LIN {X 0,Y 520.236,Z 358.517,A -85,B 0,C 180,E1 24281.743,E2 24281.743} C_VEL
LIN {X 0,Y 524.04,Z 361.624,A -85,B 0,C 180,E1 24280.378,E2 24280.378} C_VEL
LIN {X 0,Y 526.654,Z 365.44,A -85,B 0,C 180,E1 24279.437,E2 24279.437} C_VEL
LIN {X 0,Y 529.635,Z 368.07,A -85,B 0,C 180,E1 24278.486,E2 24278.486} C_VEL
LIN {X 0,Y 532.772,Z 372.256,A -85,B 0,C 180,E1 24277.489,E2 24277.489} C_VEL
LIN {X 0,Y 535.113,Z 374.487,A -85,B 0,C 180,E1 24276.809,E2 24276.809} C_VEL
LIN {X 0,Y 538.699,Z 378.866,A -85,B 0,C 180,E1 24275.782,E2 24275.782} C_VEL
LIN {X 0,Y 540.337,Z 380.709,A -85,B 0,C 180,E1 24275.336,E2 24275.336} C_VEL
LIN {X 0,Y 544.251,Z 385.306,A -85,B 0,C 180,E1 24274.305,E2 24274.305} C_VEL
LIN {X 0,Y 549.091,Z 391.188,A -85,B 0,C 180,E1 24273.095,E2 24273.095} C_VEL
LIN {X 0,Y 558.407,Z 402.895,A -85,B 0,C 180,E1 24270.941,E2 24270.941} C_VEL
LIN {X 0,Y 567.449,Z 414.718,A -85,B 0,C 180,E1 24269.034,E2 24269.034} C_VEL
LIN {X 0,Y 578.175,Z 429.194,A -85,B 0,C 180,E1 24266.962,E2 24266.962} C_VEL
LIN {X 0,Y 585.063,Z 439.312,A -85,B 0,C 180,E1 24265.711,E2 24265.711} C_VEL
LIN {X 0,Y 575.969,Z 652.824,A -85,B 0,C 180,E1 24262.521,E2 24262.521} C_VEL
LIN {X 0,Y 569.868,Z 800.136,A -85,B 0,C 180,E1 24260.332,E2 24260.332} C_VEL
LIN {X 0,Y 568.013,Z 824.85,A -85,B 0,C 180,E1 24259.864,E2 24259.864} C_VEL
LIN {X 0,Y 565.088,Z 852.733,A -85,B 0,C 180,E1 24259.144,E2 24259.144} C_VEL
LIN {X 0,Y 562.345,Z 873.984,A -85,B 0,C 180,E1 24258.454,E2 24258.454} C_VEL
LIN {X 0,Y 559.307,Z 894.579,A -85,B 0,C 180,E1 24257.656,E2 24257.656} C_VEL
LIN {X 0,Y 555.969,Z 914.69,A -85,B 0,C 180,E1 24256.747,E2 24256.747} C_VEL
LIN {X 0,Y 551.81,Z 937.435,A -85,B 0,C 180,E1 24255.554,E2 24255.554} C_VEL
LIN {X 0,Y 550.967,Z 941.891,A -85,B 0,C 180,E1 24255.296,E2 24255.296} C_VEL
LIN {X 0,Y 548.862,Z 948.783,A -85,B 0,C 180,E1 24254.955,E2 24254.955} C_VEL
LIN {X 0,Y 540.849,Z 966.119,A -85,B 0,C 180,E1 24254.291,E2 24254.291} C_VEL
LIN {X 0,Y 538.707,Z 972.514,A -85,B 0,C 180,E1 24253.919,E2 24253.919} C_VEL
LIN {X 0,Y 533.191,Z 995.822,A -85,B 0,C 180,E1 24252.097,E2 24252.097} C_VEL
LIN {X 0,Y 528.894,Z 1013.296,A -85,B 0,C 180,E1 24250.536,E2 24250.536} C_VEL
LIN {X 0,Y 524.733,Z 1029.747,A -85,B 0,C 180,E1 24248.891,E2 24248.891} C_VEL
LIN {X 0,Y 520.601,Z 1045.873,A -85,B 0,C 180,E1 24247.089,E2 24247.089} C_VEL
LIN {X 0,Y 515.835,Z 1064.561,A -85,B 0,C 180,E1 24244.741,E2 24244.741} C_VEL
LIN {X 0,Y 511.471,Z 1081.614,A -85,B 0,C 180,E1 24242.254,E2 24242.254} C_VEL
LIN {X 0,Y 508.278,Z 1094.708,A -85,B 0,C 180,E1 24240.107,E2 24240.107} C_VEL
LIN {X 0,Y 505.513,Z 1106.49,A -85,B 0,C 180,E1 24237.954,E2 24237.954} C_VEL
LIN {X 0,Y 502.961,Z 1118.198,A -85,B 0,C 180,E1 24235.555,E2 24235.555} C_VEL
LIN {X 0,Y 500.238,Z 1132.516,A -85,B 0,C 180,E1 24232.195,E2 24232.195} C_VEL
LIN {X 0,Y 498.735,Z 1141.736,A -85,B 0,C 180,E1 24229.682,E2 24229.682} C_VEL
LIN {X 0,Y 497.682,Z 1149.368,A -85,B 0,C 180,E1 24227.298,E2 24227.298} C_VEL
LIN {X 0,Y 496.911,Z 1156.239,A -85,B 0,C 180,E1 24224.806,E2 24224.806} C_VEL
LIN {X 0,Y 496.38,Z 1162.49,A -85,B 0,C 180,E1 24222.092,E2 24222.092} C_VEL
LIN {X 0,Y 496.063,Z 1168.171,A -85,B 0,C 180,E1 24218.928,E2 24218.928} C_VEL
LIN {X 0,Y 495.952,Z 1171.694,A -85,B 0,C 180,E1 24216.134,E2 24216.134} C_VEL
LIN {X 0,Y 495.915,Z 1173.799,A -85,B 0,C 180,E1 24213.578,E2 24213.578} C_VEL
LIN {X 0,Y 495.91,Z 1174.771,A -85,B 0,C 180,E1 24211.155,E2 24211.155} C_VEL
LIN {X 0,Y 495.908,Z 1174.789,A -85,B 0,C 180,E1 24208.845,E2 24208.845} C_VEL
LIN {X 0,Y 495.914,Z 1173.849,A -85,B 0,C 180,E1 24206.417,E2 24206.417} C_VEL
LIN {X 0,Y 495.949,Z 1171.784,A -85,B 0,C 180,E1 24203.866,E2 24203.866} C_VEL
LIN {X 0,Y 496.058,Z 1168.295,A -85,B 0,C 180,E1 24201.072,E2 24201.072} C_VEL
LIN {X 0,Y 496.371,Z 1162.684,A -85,B 0,C 180,E1 24197.908,E2 24197.908} C_VEL
LIN {X 0,Y 496.885,Z 1156.469,A -85,B 0,C 180,E1 24195.194,E2 24195.194} C_VEL
LIN {X 0,Y 497.652,Z 1149.635,A -85,B 0,C 180,E1 24192.701,E2 24192.701} C_VEL
LIN {X 0,Y 498.691,Z 1142.035,A -85,B 0,C 180,E1 24190.316,E2 24190.316} C_VEL
LIN {X 0,Y 500.179,Z 1132.845,A -85,B 0,C 180,E1 24187.802,E2 24187.802} C_VEL
LIN {X 0,Y 502.788,Z 1119.049,A -85,B 0,C 180,E1 24184.538,E2 24184.538} C_VEL
LIN {X 0,Y 505.406,Z 1106.924,A -85,B 0,C 180,E1 24182.04,E2 24182.04} C_VEL
LIN {X 0,Y 508.161,Z 1095.183,A -85,B 0,C 180,E1 24179.885,E2 24179.885} C_VEL
LIN {X 0,Y 511.342,Z 1082.13,A -85,B 0,C 180,E1 24177.737,E2 24177.737} C_VEL
LIN {X 0,Y 515.683,Z 1065.128,A -85,B 0,C 180,E1 24175.247,E2 24175.247} C_VEL
LIN {X 0,Y 520.505,Z 1046.256,A -85,B 0,C 180,E1 24172.865,E2 24172.865} C_VEL
LIN {X 0,Y 524.551,Z 1030.453,A -85,B 0,C 180,E1 24171.093,E2 24171.093} C_VEL
LIN {X 0,Y 528.764,Z 1013.813,A -85,B 0,C 180,E1 24169.422,E2 24169.422} C_VEL
LIN {X 0,Y 533.282,Z 995.499,A -85,B 0,C 180,E1 24167.784,E2 24167.784} C_VEL
LIN {X 0,Y 538.943,Z 971.464,A -85,B 0,C 180,E1 24165.917,E2 24165.917} C_VEL
LIN {X 0,Y 543.469,Z 950.666,A -85,B 0,C 180,E1 24164.528,E2 24164.528} C_VEL
LIN {X 0,Y 547.259,Z 931.938,A -85,B 0,C 180,E1 24163.428,E2 24163.428} C_VEL
LIN {X 0,Y 551.018,Z 911.806,A -85,B 0,C 180,E1 24162.394,E2 24162.394} C_VEL
LIN {X 0,Y 554.725,Z 889.872,A -85,B 0,C 180,E1 24161.426,E2 24161.426} C_VEL
LIN {X 0,Y 558.775,Z 861.74,A -85,B 0,C 180,E1 24160.409,E2 24160.409} C_VEL
LIN {X 0,Y 561.451,Z 839.165,A -85,B 0,C 180,E1 24159.761,E2 24159.761} C_VEL
LIN {X 0,Y 563.504,Z 817.841,A -85,B 0,C 180,E1 24159.27,E2 24159.27} C_VEL
LIN {X 0,Y 565.104,Z 795.465,A -85,B 0,C 180,E1 24158.871,E2 24158.871} C_VEL
LIN {X 0,Y 574.586,Z 574.148,A -85,B 0,C 180,E1 24155.57,E2 24155.57} C_VEL
LIN {X 0,Y 580.415,Z 443.356,A -85,B 0,C 180,E1 24153.594,E2 24153.594} C_VEL
LIN {X 0,Y 568.679,Z 426.867,A -85,B 0,C 180,E1 24151.362,E2 24151.362} C_VEL
LIN {X 0,Y 558.887,Z 413.851,A -85,B 0,C 180,E1 24149.325,E2 24149.325} C_VEL
LIN {X 0,Y 550.085,Z 402.623,A -85,B 0,C 180,E1 24147.321,E2 24147.321} C_VEL
LIN {X 0,Y 545.94,Z 397.535,A -85,B 0,C 180,E1 24146.31,E2 24146.31} C_VEL
LIN {X 0,Y 541.389,Z 391.95,A -85,B 0,C 180,E1 24145.137,E2 24145.137} C_VEL
LIN {X 0,Y 536.861,Z 386.426,A -85,B 0,C 180,E1 24143.897,E2 24143.897} C_VEL
LIN {X 0,Y 533.06,Z 381.8,A -85,B 0,C 180,E1 24142.789,E2 24142.789} C_VEL
LIN {X 0,Y 528.429,Z 376.674,A -85,B 0,C 180,E1 24141.361,E2 24141.361} C_VEL
LIN {X 0,Y 527.196,Z 374.956,A -85,B 0,C 180,E1 24140.948,E2 24140.948} C_VEL
LIN {X 0,Y 523.497,Z 371.232,A -85,B 0,C 180,E1 24139.702,E2 24139.702} C_VEL
LIN {X 0,Y 521.968,Z 368.815,A -85,B 0,C 180,E1 24139.121,E2 24139.121} C_VEL
LIN {X 0,Y 518.399,Z 365.842,A -85,B 0,C 180,E1 24137.801,E2 24137.801} C_VEL
LIN {X 0,Y 516.299,Z 362.399,A -85,B 0,C 180,E1 24136.888,E2 24136.888} C_VEL
LIN {X 0,Y 512.875,Z 359.969,A -85,B 0,C 180,E1 24135.433,E2 24135.433} C_VEL
LIN {X 0,Y 510.92,Z 356.634,A -85,B 0,C 180,E1 24134.42,E2 24134.42} C_VEL
LIN {X 0,Y 510.473,Z 355.792,A -85,B 0,C 180,E1 24134.173,E2 24134.173} C_VEL
LIN {X 0,Y 506.888,Z 353.722,A -85,B 0,C 180,E1 24132.301,E2 24132.301} C_VEL
LIN {X 0,Y 505.032,Z 350.951,A -85,B 0,C 180,E1 24131.072,E2 24131.072} C_VEL
LIN {X 0,Y 504.344,Z 349.04,A -85,B 0,C 180,E1 24130.509,E2 24130.509} C_VEL
LIN {X 0,Y 500.127,Z 346.785,A -85,B 0,C 180,E1 24127.12,E2 24127.12} C_VEL
LIN {X 0,Y 498.094,Z 343.3,A -85,B 0,C 180,E1 24124.144,E2 24124.144} C_VEL
LIN {X 0,Y 497.868,Z 342.14,A -85,B 0,C 180,E1 24123.339,E2 24123.339} C_VEL
LIN {X 0,Y 497.87,Z 342.212,A -85,B 0,C 180,E1 24119.885,E2 24119.885} C_VEL
LIN {X 0,Y 497.933,Z 342.321,A -85,B 0,C 180,E1 24116.777,E2 24116.777} C_VEL
LIN {X 0,Y 498.974,Z 345.261,A -85,B 0,C 180,E1 24114.711,E2 24114.711} C_VEL
LIN {X 0,Y 501.928,Z 348.156,A -85,B 0,C 180,E1 24111.638,E2 24111.638} C_VEL
LIN {X 0,Y 504.476,Z 349.233,A -85,B 0,C 180,E1 24109.811,E2 24109.811} C_VEL
LIN {X 0,Y 505.764,Z 352.251,A -85,B 0,C 180,E1 24108.829,E2 24108.829} C_VEL
LIN {X 0,Y 508.394,Z 354.901,A -85,B 0,C 180,E1 24107.275,E2 24107.275} C_VEL
LIN {X 0,Y 510.655,Z 356.003,A -85,B 0,C 180,E1 24106.15,E2 24106.15} C_VEL
LIN {X 0,Y 512.45,Z 359.379,A -85,B 0,C 180,E1 24105.19,E2 24105.19} C_VEL
LIN {X 0,Y 515.652,Z 362.087,A -85,B 0,C 180,E1 24103.786,E2 24103.786} C_VEL
LIN {X 0,Y 516.704,Z 362.873,A -85,B 0,C 180,E1 24103.357,E2 24103.357} C_VEL
LIN {X 0,Y 519.099,Z 366.62,A -85,B 0,C 180,E1 24102.339,E2 24102.339} C_VEL
LIN {X 0,Y 521.947,Z 369.263,A -85,B 0,C 180,E1 24101.284,E2 24101.284} C_VEL
LIN {X 0,Y 526.752,Z 375.247,A -85,B 0,C 180,E1 24099.586,E2 24099.586} C_VEL
LIN {X 0,Y 531.133,Z 380.666,A -85,B 0,C 180,E1 24098.173,E2 24098.173} C_VEL
LIN {X 0,Y 536.035,Z 386.93,A -85,B 0,C 180,E1 24096.706,E2 24096.706} C_VEL
LIN {X 0,Y 543.551,Z 396.756,A -85,B 0,C 180,E1 24094.649,E2 24094.649} C_VEL
LIN {X 0,Y 552.331,Z 408.685,A -85,B 0,C 180,E1 24092.478,E2 24092.478} C_VEL
LIN {X 0,Y 561.3,Z 421.384,A -85,B 0,C 180,E1 24090.462,E2 24090.462} C_VEL
LIN {X 0,Y 571.815,Z 437.063,A -85,B 0,C 180,E1 24088.3,E2 24088.3} C_VEL
LIN {X 0,Y 580.574,Z 450.913,A -85,B 0,C 180,E1 24086.634,E2 24086.634} C_VEL
LIN {X 0,Y 571.135,Z 666.165,A -85,B 0,C 180,E1 24083.402,E2 24083.402} C_VEL
LIN {X 0,Y 564.461,Z 823.596,A -85,B 0,C 180,E1 24081.051,E2 24081.051} C_VEL
LIN {X 0,Y 562.407,Z 849.401,A -85,B 0,C 180,E1 24080.57,E2 24080.57} C_VEL
LIN {X 0,Y 559.278,Z 877.219,A -85,B 0,C 180,E1 24079.862,E2 24079.862} C_VEL
LIN {X 0,Y 556.351,Z 898.872,A -85,B 0,C 180,E1 24079.166,E2 24079.166} C_VEL
LIN {X 0,Y 553.139,Z 919.668,A -85,B 0,C 180,E1 24078.369,E2 24078.369} C_VEL
LIN {X 0,Y 549.635,Z 940.066,A -85,B 0,C 180,E1 24077.455,E2 24077.455} C_VEL
LIN {X 0,Y 544.928,Z 965.12,A -85,B 0,C 180,E1 24076.145,E2 24076.145} C_VEL
LIN {X 0,Y 539.96,Z 988.657,A -85,B 0,C 180,E1 24074.676,E2 24074.676} C_VEL
LIN {X 0,Y 535.58,Z 1008.335,A -85,B 0,C 180,E1 24073.272,E2 24073.272} C_VEL
LIN {X 0,Y 531.279,Z 1026.905,A -85,B 0,C 180,E1 24071.776,E2 24071.776} C_VEL
LIN {X 0,Y 526.18,Z 1048.396,A -85,B 0,C 180,E1 24069.82,E2 24069.82} C_VEL
LIN {X 0,Y 521.151,Z 1068.846,A -85,B 0,C 180,E1 24067.661,E2 24067.661} C_VEL
LIN {X 0,Y 517.161,Z 1085.154,A -85,B 0,C 180,E1 24065.723,E2 24065.723} C_VEL
LIN {X 0,Y 513.478,Z 1100.386,A -85,B 0,C 180,E1 24063.708,E2 24063.708} C_VEL
LIN {X 0,Y 509.457,Z 1117.58,A -85,B 0,C 180,E1 24061.16,E2 24061.16} C_VEL
LIN {X 0,Y 505.895,Z 1133.58,A -85,B 0,C 180,E1 24058.413,E2 24058.413} C_VEL
LIN {X 0,Y 503.341,Z 1145.834,A -85,B 0,C 180,E1 24056.04,E2 24056.04} C_VEL
LIN {X 0,Y 501.539,Z 1155.249,A -85,B 0,C 180,E1 24053.997,E2 24053.997} C_VEL
LIN {X 0,Y 499.8,Z 1164.972,A -85,B 0,C 180,E1 24051.598,E2 24051.598} C_VEL
LIN {X 0,Y 498.43,Z 1173.911,A -85,B 0,C 180,E1 24049.086,E2 24049.086} C_VEL
LIN {X 0,Y 497.194,Z 1183.627,A -85,B 0,C 180,E1 24045.872,E2 24045.872} C_VEL
LIN {X 0,Y 496.525,Z 1190.553,A -85,B 0,C 180,E1 24043.034,E2 24043.034} C_VEL
LIN {X 0,Y 496.175,Z 1195.689,A -85,B 0,C 180,E1 24040.448,E2 24040.448} C_VEL
LIN {X 0,Y 496.01,Z 1199.512,A -85,B 0,C 180,E1 24037.995,E2 24037.995} C_VEL
LIN {X 0,Y 495.933,Z 1202.422,A -85,B 0,C 180,E1 24035.437,E2 24035.437} C_VEL
LIN {X 0,Y 495.91,Z 1204.435,A -85,B 0,C 180,E1 24032.542,E2 24032.542} C_VEL
LIN {X 0,Y 495.896,Z 1204.894,A -85,B 0,C 180,E1 24029.422,E2 24029.422} C_VEL
LIN {X 0,Y 495.916,Z 1204.094,A -85,B 0,C 180,E1 24026.879,E2 24026.879} C_VEL
LIN {X 0,Y 495.937,Z 1202.193,A -85,B 0,C 180,E1 24024.331,E2 24024.331} C_VEL
LIN {X 0,Y 496.015,Z 1199.351,A -85,B 0,C 180,E1 24021.888,E2 24021.888} C_VEL
LIN {X 0,Y 496.186,Z 1195.48,A -85,B 0,C 180,E1 24019.434,E2 24019.434} C_VEL
LIN {X 0,Y 496.551,Z 1190.298,A -85,B 0,C 180,E1 24016.848,E2 24016.848} C_VEL
LIN {X 0,Y 497.298,Z 1182.679,A -85,B 0,C 180,E1 24013.771,E2 24013.771} C_VEL
LIN {X 0,Y 498.488,Z 1173.505,A -85,B 0,C 180,E1 24010.795,E2 24010.795} C_VEL
LIN {X 0,Y 499.8,Z 1164.976,A -85,B 0,C 180,E1 24008.402,E2 24008.402} C_VEL
LIN {X 0,Y 501.541,Z 1155.256,A -85,B 0,C 180,E1 24006.003,E2 24006.003} C_VEL
LIN {X 0,Y 503.459,Z 1145.256,A -85,B 0,C 180,E1 24003.84,E2 24003.84} C_VEL
LIN {X 0,Y 506.258,Z 1131.902,A -85,B 0,C 180,E1 24001.274,E2 24001.274} C_VEL
LIN {X 0,Y 510.053,Z 1114.954,A -85,B 0,C 180,E1 23998.439,E2 23998.439} C_VEL
LIN {X 0,Y 513.572,Z 1099.989,A -85,B 0,C 180,E1 23996.237,E2 23996.237} C_VEL
LIN {X 0,Y 517.161,Z 1085.156,A -85,B 0,C 180,E1 23994.277,E2 23994.277} C_VEL
LIN {X 0,Y 521.151,Z 1068.847,A -85,B 0,C 180,E1 23992.339,E2 23992.339} C_VEL
LIN {X 0,Y 526.283,Z 1047.928,A -85,B 0,C 180,E1 23990.136,E2 23990.136} C_VEL
LIN {X 0,Y 531.276,Z 1026.894,A -85,B 0,C 180,E1 23988.224,E2 23988.224} C_VEL
LIN {X 0,Y 535.576,Z 1008.328,A -85,B 0,C 180,E1 23986.728,E2 23986.728} C_VEL
LIN {X 0,Y 539.957,Z 988.648,A -85,B 0,C 180,E1 23985.324,E2 23985.324} C_VEL
LIN {X 0,Y 545.113,Z 964.104,A -85,B 0,C 180,E1 23983.8,E2 23983.8} C_VEL
LIN {X 0,Y 549.63,Z 940.037,A -85,B 0,C 180,E1 23982.545,E2 23982.545} C_VEL
LIN {X 0,Y 553.133,Z 919.623,A -85,B 0,C 180,E1 23981.63,E2 23981.63} C_VEL
LIN {X 0,Y 556.346,Z 898.815,A -85,B 0,C 180,E1 23980.833,E2 23980.833} C_VEL
LIN {X 0,Y 559.316,Z 876.821,A -85,B 0,C 180,E1 23980.128,E2 23980.128} C_VEL
LIN {X 0,Y 562.476,Z 848.4,A -85,B 0,C 180,E1 23979.411,E2 23979.411} C_VEL
LIN {X 0,Y 564.452,Z 823.42,A -85,B 0,C 180,E1 23978.948,E2 23978.948} C_VEL
LIN {X 0,Y 572.713,Z 628.453,A -85,B 0,C 180,E1 23976.039,E2 23976.039} C_VEL
LIN {X 0,Y 580.49,Z 450.828,A -85,B 0,C 180,E1 23973.361,E2 23973.361} C_VEL
LIN {X 0,Y 571.078,Z 436.028,A -85,B 0,C 180,E1 23971.568,E2 23971.568} C_VEL
LIN {X 0,Y 560.599,Z 420.343,A -85,B 0,C 180,E1 23969.402,E2 23969.402} C_VEL
LIN {X 0,Y 549.949,Z 405.419,A -85,B 0,C 180,E1 23966.977,E2 23966.977} C_VEL
LIN {X 0,Y 541.131,Z 393.611,A -85,B 0,C 180,E1 23964.741,E2 23964.741} C_VEL
LIN {X 0,Y 534.034,Z 384.385,A -85,B 0,C 180,E1 23962.746,E2 23962.746} C_VEL
LIN {X 0,Y 529.555,Z 378.709,A -85,B 0,C 180,E1 23961.372,E2 23961.372} C_VEL
LIN {X 0,Y 524.876,Z 372.97,A -85,B 0,C 180,E1 23959.822,E2 23959.822} C_VEL
LIN {X 0,Y 521.1,Z 368.313,A -85,B 0,C 180,E1 23958.458,E2 23958.458} C_VEL
LIN {X 0,Y 518.032,Z 365.287,A -85,B 0,C 180,E1 23957.292,E2 23957.292} C_VEL
LIN {X 0,Y 516.304,Z 362.402,A -85,B 0,C 180,E1 23956.54,E2 23956.54} C_VEL
LIN {X 0,Y 512.868,Z 359.866,A -85,B 0,C 180,E1 23955.086,E2 23955.086} C_VEL
LIN {X 0,Y 510.836,Z 356.524,A -85,B 0,C 180,E1 23954.047,E2 23954.047} C_VEL
LIN {X 0,Y 510.437,Z 355.759,A -85,B 0,C 180,E1 23953.827,E2 23953.827} C_VEL
LIN {X 0,Y 507.013,Z 353.838,A -85,B 0,C 180,E1 23952.066,E2 23952.066} C_VEL
LIN {X 0,Y 504.889,Z 350.566,A -85,B 0,C 180,E1 23950.671,E2 23950.671} C_VEL
LIN {X 0,Y 504.421,Z 349.043,A -85,B 0,C 180,E1 23950.277,E2 23950.277} C_VEL
LIN {X 0,Y 500.434,Z 347.063,A -85,B 0,C 180,E1 23947.231,E2 23947.231} C_VEL
LIN {X 0,Y 498.21,Z 343.675,A -85,B 0,C 180,E1 23944.374,E2 23944.374} C_VEL
LIN {X 0,Y 497.91,Z 342.135,A -85,B 0,C 180,E1 23943.569,E2 23943.569} C_VEL
LIN {X 0,Y 497.875,Z 342.216,A -85,B 0,C 180,E1 23940.115,E2 23940.115} C_VEL
LIN {X 0,Y 497.865,Z 342.141,A -85,B 0,C 180,E1 23936.484,E2 23936.484} C_VEL
LIN {X 0,Y 497.918,Z 342.459,A -85,B 0,C 180,E1 23935.797,E2 23935.797} C_VEL
LIN {X 0,Y 499.239,Z 345.748,A -85,B 0,C 180,E1 23933.56,E2 23933.56} C_VEL
LIN {X 0,Y 502.845,Z 348.594,A -85,B 0,C 180,E1 23930.269,E2 23930.269} C_VEL
LIN {X 0,Y 504.501,Z 349.313,A -85,B 0,C 180,E1 23929.147,E2 23929.147} C_VEL
LIN {X 0,Y 505.68,Z 352.253,A -85,B 0,C 180,E1 23928.249,E2 23928.249} C_VEL
LIN {X 0,Y 508.557,Z 354.98,A -85,B 0,C 180,E1 23926.585,E2 23926.585} C_VEL
LIN {X 0,Y 510.678,Z 356.028,A -85,B 0,C 180,E1 23925.544,E2 23925.544} C_VEL
LIN {X 0,Y 512.428,Z 359.427,A -85,B 0,C 180,E1 23924.611,E2 23924.611} C_VEL
LIN {X 0,Y 515.393,Z 361.958,A -85,B 0,C 180,E1 23923.314,E2 23923.314} C_VEL
LIN {X 0,Y 516.584,Z 362.81,A -85,B 0,C 180,E1 23922.832,E2 23922.832} C_VEL
LIN {X 0,Y 518.994,Z 366.518,A -85,B 0,C 180,E1 23921.814,E2 23921.814} C_VEL
LIN {X 0,Y 522.327,Z 369.303,A -85,B 0,C 180,E1 23920.602,E2 23920.602} C_VEL
LIN {X 0,Y 525.385,Z 373.462,A -85,B 0,C 180,E1 23919.501,E2 23919.501} C_VEL
LIN {X 0,Y 527.855,Z 375.748,A -85,B 0,C 180,E1 23918.702,E2 23918.702} C_VEL
LIN {X 0,Y 531.312,Z 380.127,A -85,B 0,C 180,E1 23917.599,E2 23917.599} C_VEL
LIN {X 0,Y 533.271,Z 382.147,A -85,B 0,C 180,E1 23917.018,E2 23917.018} C_VEL
LIN {X 0,Y 537.21,Z 386.738,A -85,B 0,C 180,E1 23915.886,E2 23915.886} C_VEL
LIN {X 0,Y 542.151,Z 392.676,A -85,B 0,C 180,E1 23914.55,E2 23914.55} C_VEL
LIN {X 0,Y 546.944,Z 398.552,A -85,B 0,C 180,E1 23913.333,E2 23913.333} C_VEL
LIN {X 0,Y 556.267,Z 410.523,A -85,B 0,C 180,E1 23911.143,E2 23911.143} C_VEL
LIN {X 0,Y 564.469,Z 421.296,A -85,B 0,C 180,E1 23909.384,E2 23909.384} C_VEL
LIN {X 0,Y 575.542,Z 436.424,A -85,B 0,C 180,E1 23907.207,E2 23907.207} C_VEL
LIN {X 0,Y 580.401,Z 443.667,A -85,B 0,C 180,E1 23906.303,E2 23906.303} C_VEL
LIN {X 0,Y 570.968,Z 656.962,A -85,B 0,C 180,E1 23903.101,E2 23903.101} C_VEL
LIN {X 0,Y 564.79,Z 800.458,A -85,B 0,C 180,E1 23900.956,E2 23900.956} C_VEL
LIN {X 0,Y 562.856,Z 825.404,A -85,B 0,C 180,E1 23900.482,E2 23900.482} C_VEL
LIN {X 0,Y 559.848,Z 853.118,A -85,B 0,C 180,E1 23899.763,E2 23899.763} C_VEL
LIN {X 0,Y 556.979,Z 874.623,A -85,B 0,C 180,E1 23899.061,E2 23899.061} C_VEL
LIN {X 0,Y 553.916,Z 894.727,A -85,B 0,C 180,E1 23898.279,E2 23898.279} C_VEL
LIN {X 0,Y 550.349,Z 915.483,A -85,B 0,C 180,E1 23897.337,E2 23897.337} C_VEL
LIN {X 0,Y 545.768,Z 939.703,A -85,B 0,C 180,E1 23896.053,E2 23896.053} C_VEL
LIN {X 0,Y 540.731,Z 963.237,A -85,B 0,C 180,E1 23894.566,E2 23894.566} C_VEL
LIN {X 0,Y 538.707,Z 972.514,A -85,B 0,C 180,E1 23893.919,E2 23893.919} C_VEL
LIN {X 0,Y 536.517,Z 978.993,A -85,B 0,C 180,E1 23893.526,E2 23893.526} C_VEL
LIN {X 0,Y 528.001,Z 995.476,A -85,B 0,C 180,E1 23892.675,E2 23892.675} C_VEL
LIN {X 0,Y 525.705,Z 1001.573,A -85,B 0,C 180,E1 23892.226,E2 23892.226} C_VEL
LIN {X 0,Y 520.245,Z 1022.906,A -85,B 0,C 180,E1 23890.222,E2 23890.222} C_VEL
LIN {X 0,Y 515.074,Z 1042.157,A -85,B 0,C 180,E1 23888.119,E2 23888.119} C_VEL
LIN {X 0,Y 510.918,Z 1057.554,A -85,B 0,C 180,E1 23886.228,E2 23886.228} C_VEL
LIN {X 0,Y 507.147,Z 1071.643,A -85,B 0,C 180,E1 23884.299,E2 23884.299} C_VEL
LIN {X 0,Y 503.464,Z 1085.677,A -85,B 0,C 180,E1 23882.157,E2 23882.157} C_VEL
LIN {X 0,Y 499.39,Z 1101.788,A -85,B 0,C 180,E1 23879.375,E2 23879.375} C_VEL
LIN {X 0,Y 496.221,Z 1115.105,A -85,B 0,C 180,E1 23876.701,E2 23876.701} C_VEL
LIN {X 0,Y 493.89,Z 1125.827,A -85,B 0,C 180,E1 23874.265,E2 23874.265} C_VEL
LIN {X 0,Y 492.03,Z 1135.294,A -85,B 0,C 180,E1 23871.831,E2 23871.831} C_VEL
LIN {X 0,Y 490.343,Z 1145.785,A -85,B 0,C 180,E1 23868.795,E2 23868.795} C_VEL
LIN {X 0,Y 489.167,Z 1154.722,A -85,B 0,C 180,E1 23865.653,E2 23865.653} C_VEL
LIN {X 0,Y 488.537,Z 1160.963,A -85,B 0,C 180,E1 23863.01,E2 23863.01} C_VEL
LIN {X 0,Y 488.194,Z 1165.812,A -85,B 0,C 180,E1 23860.502,E2 23860.502} C_VEL
LIN {X 0,Y 488.016,Z 1169.607,A -85,B 0,C 180,E1 23858.008,E2 23858.008} C_VEL
LIN {X 0,Y 487.932,Z 1172.488,A -85,B 0,C 180,E1 23855.409,E2 23855.409} C_VEL
LIN {X 0,Y 487.908,Z 1174.529,A -85,B 0,C 180,E1 23852.349,E2 23852.349} C_VEL
LIN {X 0,Y 487.898,Z 1174.88,A -85,B 0,C 180,E1 23849.295,E2 23849.295} C_VEL
LIN {X 0,Y 487.912,Z 1174.05,A -85,B 0,C 180,E1 23846.711,E2 23846.711} C_VEL
LIN {X 0,Y 487.939,Z 1172.235,A -85,B 0,C 180,E1 23844.237,E2 23844.237} C_VEL
LIN {X 0,Y 488.027,Z 1169.374,A -85,B 0,C 180,E1 23841.728,E2 23841.728} C_VEL
LIN {X 0,Y 488.205,Z 1165.555,A -85,B 0,C 180,E1 23839.259,E2 23839.259} C_VEL
LIN {X 0,Y 488.598,Z 1160.39,A -85,B 0,C 180,E1 23836.63,E2 23836.63} C_VEL
LIN {X 0,Y 489.392,Z 1152.808,A -85,B 0,C 180,E1 23833.502,E2 23833.502} C_VEL
LIN {X 0,Y 490.647,Z 1143.652,A -85,B 0,C 180,E1 23830.476,E2 23830.476} C_VEL
LIN {X 0,Y 492.222,Z 1134.266,A -85,B 0,C 180,E1 23827.801,E2 23827.801} C_VEL
LIN {X 0,Y 494.233,Z 1124.162,A -85,B 0,C 180,E1 23825.243,E2 23825.243} C_VEL
LIN {X 0,Y 497.333,Z 1110.308,A -85,B 0,C 180,E1 23822.198,E2 23822.198} C_VEL
LIN {X 0,Y 500.633,Z 1096.75,A -85,B 0,C 180,E1 23819.634,E2 23819.634} C_VEL
LIN {X 0,Y 503.904,Z 1083.914,A -85,B 0,C 180,E1 23817.471,E2 23817.471} C_VEL
LIN {X 0,Y 507.473,Z 1070.386,A -85,B 0,C 180,E1 23815.428,E2 23815.428} C_VEL
LIN {X 0,Y 512.006,Z 1053.586,A -85,B 0,C 180,E1 23813.165,E2 23813.165} C_VEL
LIN {X 0,Y 517.43,Z 1033.343,A -85,B 0,C 180,E1 23810.796,E2 23810.796} C_VEL
LIN {X 0,Y 521.878,Z 1016.482,A -85,B 0,C 180,E1 23809.063,E2 23809.063} C_VEL
LIN {X 0,Y 526.393,Z 998.904,A -85,B 0,C 180,E1 23807.452,E2 23807.452} C_VEL
LIN {X 0,Y 531.06,Z 980.034,A -85,B 0,C 180,E1 23805.919,E2 23805.919} C_VEL
LIN {X 0,Y 536.817,Z 955.391,A -85,B 0,C 180,E1 23804.186,E2 23804.186} C_VEL
LIN {X 0,Y 541.294,Z 934.192,A -85,B 0,C 180,E1 23802.912,E2 23802.912} C_VEL
LIN {X 0,Y 545.165,Z 914.308,A -85,B 0,C 180,E1 23801.874,E2 23801.874} C_VEL
LIN {X 0,Y 548.546,Z 895.233,A -85,B 0,C 180,E1 23801.009,E2 23801.009} C_VEL
LIN {X 0,Y 551.825,Z 874.442,A -85,B 0,C 180,E1 23800.199,E2 23800.199} C_VEL
LIN {X 0,Y 555.076,Z 850.656,A -85,B 0,C 180,E1 23799.429,E2 23799.429} C_VEL
LIN {X 0,Y 558.081,Z 822.454,A -85,B 0,C 180,E1 23798.723,E2 23798.723} C_VEL
LIN {X 0,Y 559.878,Z 799.571,A -85,B 0,C 180,E1 23798.296,E2 23798.296} C_VEL
LIN {X 0,Y 569.203,Z 591.089,A -85,B 0,C 180,E1 23795.167,E2 23795.167} C_VEL
LIN {X 0,Y 575.765,Z 447.836,A -85,B 0,C 180,E1 23792.986,E2 23792.986} C_VEL
LIN {X 0,Y 565.116,Z 432.652,A -85,B 0,C 180,E1 23790.901,E2 23790.901} C_VEL
LIN {X 0,Y 555.679,Z 420.101,A -85,B 0,C 180,E1 23788.891,E2 23788.891} C_VEL
LIN {X 0,Y 547.618,Z 409.649,A -85,B 0,C 180,E1 23787.013,E2 23787.013} C_VEL
LIN {X 0,Y 543.33,Z 404.368,A -85,B 0,C 180,E1 23785.947,E2 23785.947} C_VEL
LIN {X 0,Y 539.124,Z 399.122,A -85,B 0,C 180,E1 23784.84,E2 23784.84} C_VEL
LIN {X 0,Y 534.653,Z 393.631,A -85,B 0,C 180,E1 23783.592,E2 23783.592} C_VEL
LIN {X 0,Y 530.064,Z 388.145,A -85,B 0,C 180,E1 23782.223,E2 23782.223} C_VEL
LIN {X 0,Y 526.282,Z 383.698,A -85,B 0,C 180,E1 23781.015,E2 23781.015} C_VEL
LIN {X 0,Y 525.123,Z 382.294,A -85,B 0,C 180,E1 23780.626,E2 23780.626} C_VEL
LIN {X 0,Y 521.441,Z 378.283,A -85,B 0,C 180,E1 23779.345,E2 23779.345} C_VEL
LIN {X 0,Y 520.128,Z 376.353,A -85,B 0,C 180,E1 23778.842,E2 23778.842} C_VEL
LIN {X 0,Y 516.637,Z 373.217,A -85,B 0,C 180,E1 23777.515,E2 23777.515} C_VEL
LIN {X 0,Y 514.815,Z 370.16,A -85,B 0,C 180,E1 23776.705,E2 23776.705} C_VEL
LIN {X 0,Y 511.442,Z 367.658,A -85,B 0,C 180,E1 23775.245,E2 23775.245} C_VEL
LIN {X 0,Y 509.313,Z 364.016,A -85,B 0,C 180,E1 23774.119,E2 23774.119} C_VEL
LIN {X 0,Y 508.386,Z 363.363,A -85,B 0,C 180,E1 23773.652,E2 23773.652} C_VEL
LIN {X 0,Y 504.835,Z 360.625,A -85,B 0,C 180,E1 23771.655,E2 23771.655} C_VEL
LIN {X 0,Y 503.288,Z 357.422,A -85,B 0,C 180,E1 23770.503,E2 23770.503} C_VEL
LIN {X 0,Y 502.87,Z 356.873,A -85,B 0,C 180,E1 23770.193,E2 23770.193} C_VEL
LIN {X 0,Y 498.944,Z 354.543,A -85,B 0,C 180,E1 23766.906,E2 23766.906} C_VEL
LIN {X 0,Y 497.062,Z 351.182,A -85,B 0,C 180,E1 23764.037,E2 23764.037} C_VEL
LIN {X 0,Y 496.78,Z 350.063,A -85,B 0,C 180,E1 23763.231,E2 23763.231} C_VEL
LIN {X 0,Y 496.906,Z 350.216,A -85,B 0,C 180,E1 23756.886,E2 23756.886} C_VEL
LIN {X 0,Y 497.916,Z 353.139,A -85,B 0,C 180,E1 23754.815,E2 23754.815} C_VEL
LIN {X 0,Y 500.822,Z 356.043,A -85,B 0,C 180,E1 23751.735,E2 23751.735} C_VEL
LIN {X 0,Y 503.202,Z 357.18,A -85,B 0,C 180,E1 23749.987,E2 23749.987} C_VEL
LIN {X 0,Y 504.78,Z 360.426,A -85,B 0,C 180,E1 23748.806,E2 23748.806} C_VEL
LIN {X 0,Y 507.437,Z 362.898,A -85,B 0,C 180,E1 23747.25,E2 23747.25} C_VEL
LIN {X 0,Y 509.233,Z 363.883,A -85,B 0,C 180,E1 23746.343,E2 23746.343} C_VEL
LIN {X 0,Y 511.359,Z 367.473,A -85,B 0,C 180,E1 23745.216,E2 23745.216} C_VEL
LIN {X 0,Y 515.143,Z 370.63,A -85,B 0,C 180,E1 23743.567,E2 23743.567} C_VEL
LIN {X 0,Y 517.859,Z 374.597,A -85,B 0,C 180,E1 23742.412,E2 23742.412} C_VEL
LIN {X 0,Y 520.261,Z 376.826,A -85,B 0,C 180,E1 23741.511,E2 23741.511} C_VEL
LIN {X 0,Y 525.003,Z 382.828,A -85,B 0,C 180,E1 23739.806,E2 23739.806} C_VEL
LIN {X 0,Y 529.251,Z 388.167,A -85,B 0,C 180,E1 23738.412,E2 23738.412} C_VEL
LIN {X 0,Y 534.011,Z 394.317,A -85,B 0,C 180,E1 23736.962,E2 23736.962} C_VEL
LIN {X 0,Y 541.346,Z 404.043,A -85,B 0,C 180,E1 23734.919,E2 23734.919} C_VEL
LIN {X 0,Y 550.432,Z 416.532,A -85,B 0,C 180,E1 23732.639,E2 23732.639} C_VEL
LIN {X 0,Y 559.972,Z 430.331,A -85,B 0,C 180,E1 23730.473,E2 23730.473} C_VEL
LIN {X 0,Y 570.34,Z 446.124,A -85,B 0,C 180,E1 23728.327,E2 23728.327} C_VEL
LIN {X 0,Y 575.955,Z 455.358,A -85,B 0,C 180,E1 23727.232,E2 23727.232} C_VEL
LIN {X 0,Y 566.218,Z 669.367,A -85,B 0,C 180,E1 23724.004,E2 23724.004} C_VEL
LIN {X 0,Y 559.434,Z 823.349,A -85,B 0,C 180,E1 23721.692,E2 23721.692} C_VEL
LIN {X 0,Y 557.308,Z 849.313,A -85,B 0,C 180,E1 23721.207,E2 23721.207} C_VEL
LIN {X 0,Y 554.093,Z 876.962,A -85,B 0,C 180,E1 23720.502,E2 23720.502} C_VEL
LIN {X 0,Y 551.068,Z 898.613,A -85,B 0,C 180,E1 23719.806,E2 23719.806} C_VEL
LIN {X 0,Y 547.746,Z 919.406,A -85,B 0,C 180,E1 23719.008,E2 23719.008} C_VEL
LIN {X 0,Y 544.122,Z 939.802,A -85,B 0,C 180,E1 23718.091,E2 23718.091} C_VEL
LIN {X 0,Y 539.247,Z 964.854,A -85,B 0,C 180,E1 23716.776,E2 23716.776} C_VEL
LIN {X 0,Y 534.018,Z 988.721,A -85,B 0,C 180,E1 23715.279,E2 23715.279} C_VEL
LIN {X 0,Y 529.488,Z 1008.324,A -85,B 0,C 180,E1 23713.87,E2 23713.87} C_VEL
LIN {X 0,Y 524.993,Z 1026.966,A -85,B 0,C 180,E1 23712.355,E2 23712.355} C_VEL
LIN {X 0,Y 519.61,Z 1048.704,A -85,B 0,C 180,E1 23710.356,E2 23710.356} C_VEL
LIN {X 0,Y 514.366,Z 1069.042,A -85,B 0,C 180,E1 23708.181,E2 23708.181} C_VEL
LIN {X 0,Y 510.251,Z 1085.136,A -85,B 0,C 180,E1 23706.245,E2 23706.245} C_VEL
LIN {X 0,Y 506.456,Z 1100.108,A -85,B 0,C 180,E1 23704.239,E2 23704.239} C_VEL
LIN {X 0,Y 502.318,Z 1117.027,A -85,B 0,C 180,E1 23701.701,E2 23701.701} C_VEL
LIN {X 0,Y 498.513,Z 1133.144,A -85,B 0,C 180,E1 23698.906,E2 23698.906} C_VEL
LIN {X 0,Y 495.795,Z 1145.558,A -85,B 0,C 180,E1 23696.467,E2 23696.467} C_VEL
LIN {X 0,Y 493.69,Z 1156.076,A -85,B 0,C 180,E1 23694.149,E2 23694.149} C_VEL
LIN {X 0,Y 491.913,Z 1165.888,A -85,B 0,C 180,E1 23691.711,E2 23691.711} C_VEL
LIN {X 0,Y 490.276,Z 1176.321,A -85,B 0,C 180,E1 23688.674,E2 23688.674} C_VEL
LIN {X 0,Y 489.153,Z 1184.836,A -85,B 0,C 180,E1 23685.653,E2 23685.653} C_VEL
LIN {X 0,Y 488.553,Z 1190.804,A -85,B 0,C 180,E1 23683.13,E2 23683.13} C_VEL
LIN {X 0,Y 488.196,Z 1195.684,A -85,B 0,C 180,E1 23680.622,E2 23680.622} C_VEL
LIN {X 0,Y 488.017,Z 1199.509,A -85,B 0,C 180,E1 23678.127,E2 23678.127} C_VEL
LIN {X 0,Y 487.937,Z 1202.305,A -85,B 0,C 180,E1 23675.645,E2 23675.645} C_VEL
LIN {X 0,Y 487.914,Z 1204.228,A -85,B 0,C 180,E1 23672.937,E2 23672.937} C_VEL
LIN {X 0,Y 487.9,Z 1204.961,A -85,B 0,C 180,E1 23669.765,E2 23669.765} C_VEL
LIN {X 0,Y 487.916,Z 1204.091,A -85,B 0,C 180,E1 23666.828,E2 23666.828} C_VEL
LIN {X 0,Y 487.939,Z 1202.19,A -85,B 0,C 180,E1 23664.237,E2 23664.237} C_VEL
LIN {X 0,Y 488.022,Z 1199.318,A -85,B 0,C 180,E1 23661.732,E2 23661.732} C_VEL
LIN {X 0,Y 488.206,Z 1195.477,A -85,B 0,C 180,E1 23659.259,E2 23659.259} C_VEL
LIN {X 0,Y 488.605,Z 1190.295,A -85,B 0,C 180,E1 23656.63,E2 23656.63} C_VEL
LIN {X 0,Y 489.406,Z 1182.678,A -85,B 0,C 180,E1 23653.502,E2 23653.502} C_VEL
LIN {X 0,Y 490.674,Z 1173.504,A -85,B 0,C 180,E1 23650.477,E2 23650.477} C_VEL
LIN {X 0,Y 492.077,Z 1164.966,A -85,B 0,C 180,E1 23648.045,E2 23648.045} C_VEL
LIN {X 0,Y 493.889,Z 1155.031,A -85,B 0,C 180,E1 23645.607,E2 23645.607} C_VEL
LIN {X 0,Y 496.185,Z 1143.81,A -85,B 0,C 180,E1 23643.168,E2 23643.168} C_VEL
LIN {X 0,Y 499.588,Z 1128.516,A -85,B 0,C 180,E1 23640.242,E2 23640.242} C_VEL
LIN {X 0,Y 503.247,Z 1113.109,A -85,B 0,C 180,E1 23637.693,E2 23637.693} C_VEL
LIN {X 0,Y 506.807,Z 1098.658,A -85,B 0,C 180,E1 23635.557,E2 23635.557} C_VEL
LIN {X 0,Y 510.791,Z 1082.998,A -85,B 0,C 180,E1 23633.482,E2 23633.482} C_VEL
LIN {X 0,Y 516.011,Z 1062.79,A -85,B 0,C 180,E1 23631.112,E2 23631.112} C_VEL
LIN {X 0,Y 520.963,Z 1043.19,A -85,B 0,C 180,E1 23629.121,E2 23629.121} C_VEL
LIN {X 0,Y 525.407,Z 1025.267,A -85,B 0,C 180,E1 23627.502,E2 23627.502} C_VEL
LIN {X 0,Y 529.846,Z 1006.816,A -85,B 0,C 180,E1 23626.017,E2 23626.017} C_VEL
LIN {X 0,Y 534.804,Z 985.357,A -85,B 0,C 180,E1 23624.495,E2 23624.495} C_VEL
LIN {X 0,Y 540.241,Z 959.776,A -85,B 0,C 180,E1 23622.948,E2 23622.948} C_VEL
LIN {X 0,Y 544.326,Z 938.622,A -85,B 0,C 180,E1 23621.854,E2 23621.854} C_VEL
LIN {X 0,Y 547.957,Z 918.056,A -85,B 0,C 180,E1 23620.938,E2 23620.938} C_VEL
LIN {X 0,Y 551.286,Z 897.053,A -85,B 0,C 180,E1 23620.141,E2 23620.141} C_VEL
LIN {X 0,Y 554.958,Z 870.498,A -85,B 0,C 180,E1 23619.312,E2 23619.312} C_VEL
LIN {X 0,Y 557.735,Z 844.278,A -85,B 0,C 180,E1 23618.694,E2 23618.694} C_VEL
LIN {X 0,Y 559.513,Z 821.634,A -85,B 0,C 180,E1 23618.282,E2 23618.282} C_VEL
LIN {X 0,Y 568.788,Z 610.555,A -85,B 0,C 180,E1 23615.116,E2 23615.116} C_VEL
LIN {X 0,Y 575.874,Z 454.996,A -85,B 0,C 180,E1 23612.757,E2 23612.757} C_VEL
LIN {X 0,Y 564.913,Z 437.802,A -85,B 0,C 180,E1 23610.589,E2 23610.589} C_VEL
LIN {X 0,Y 556.614,Z 425.504,A -85,B 0,C 180,E1 23608.808,E2 23608.808} C_VEL
LIN {X 0,Y 547.474,Z 412.435,A -85,B 0,C 180,E1 23606.669,E2 23606.669} C_VEL
LIN {X 0,Y 538.68,Z 400.519,A -85,B 0,C 180,E1 23604.394,E2 23604.394} C_VEL
LIN {X 0,Y 532.034,Z 391.747,A -85,B 0,C 180,E1 23602.486,E2 23602.486} C_VEL
LIN {X 0,Y 527.45,Z 385.914,A -85,B 0,C 180,E1 23601.053,E2 23601.053} C_VEL
LIN {X 0,Y 523.001,Z 380.344,A -85,B 0,C 180,E1 23599.547,E2 23599.547} C_VEL
LIN {X 0,Y 519.417,Z 375.916,A -85,B 0,C 180,E1 23598.229,E2 23598.229} C_VEL
LIN {X 0,Y 516.271,Z 372.648,A -85,B 0,C 180,E1 23597.005,E2 23597.005} C_VEL
LIN {X 0,Y 514.816,Z 370.159,A -85,B 0,C 180,E1 23596.357,E2 23596.357} C_VEL
LIN {X 0,Y 511.316,Z 367.421,A -85,B 0,C 180,E1 23594.843,E2 23594.843} C_VEL
LIN {X 0,Y 509.223,Z 363.899,A -85,B 0,C 180,E1 23593.744,E2 23593.744} C_VEL
LIN {X 0,Y 505.208,Z 361.026,A -85,B 0,C 180,E1 23591.589,E2 23591.589} C_VEL
LIN {X 0,Y 503.303,Z 357.543,A -85,B 0,C 180,E1 23590.242,E2 23590.242} C_VEL
LIN {X 0,Y 502.936,Z 356.865,A -85,B 0,C 180,E1 23589.96,E2 23589.96} C_VEL
LIN {X 0,Y 499.003,Z 354.649,A -85,B 0,C 180,E1 23586.79,E2 23586.79} C_VEL
LIN {X 0,Y 496.962,Z 350.768,A -85,B 0,C 180,E1 23583.807,E2 23583.807} C_VEL
LIN {X 0,Y 496.783,Z 350.052,A -85,B 0,C 180,E1 23583.346,E2 23583.346} C_VEL
LIN {X 0,Y 496.819,Z 350.079,A -85,B 0,C 180,E1 23576.076,E2 23576.076} C_VEL
LIN {X 0,Y 498.17,Z 353.626,A -85,B 0,C 180,E1 23573.662,E2 23573.662} C_VEL
LIN {X 0,Y 501.726,Z 356.486,A -85,B 0,C 180,E1 23570.363,E2 23570.363} C_VEL
LIN {X 0,Y 503.188,Z 357.178,A -85,B 0,C 180,E1 23569.35,E2 23569.35} C_VEL
LIN {X 0,Y 504.611,Z 360.322,A -85,B 0,C 180,E1 23568.281,E2 23568.281} C_VEL
LIN {X 0,Y 508.034,Z 363.206,A -85,B 0,C 180,E1 23566.339,E2 23566.339} C_VEL
LIN {X 0,Y 509.251,Z 363.934,A -85,B 0,C 180,E1 23565.735,E2 23565.735} C_VEL
LIN {X 0,Y 511.336,Z 367.543,A -85,B 0,C 180,E1 23564.635,E2 23564.635} C_VEL
LIN {X 0,Y 515.022,Z 370.571,A -85,B 0,C 180,E1 23563.04,E2 23563.04} C_VEL
LIN {X 0,Y 517.62,Z 374.352,A -85,B 0,C 180,E1 23561.938,E2 23561.938} C_VEL
LIN {X 0,Y 520.693,Z 377.065,A -85,B 0,C 180,E1 23560.801,E2 23560.801} C_VEL
LIN {X 0,Y 523.964,Z 381.309,A -85,B 0,C 180,E1 23559.618,E2 23559.618} C_VEL
LIN {X 0,Y 526.087,Z 383.392,A -85,B 0,C 180,E1 23558.919,E2 23558.919} C_VEL
LIN {X 0,Y 529.856,Z 387.981,A -85,B 0,C 180,E1 23557.709,E2 23557.709} C_VEL
LIN {X 0,Y 531.533,Z 389.92,A -85,B 0,C 180,E1 23557.2,E2 23557.2} C_VEL
LIN {X 0,Y 536.399,Z 395.783,A -85,B 0,C 180,E1 23555.789,E2 23555.789} C_VEL
LIN {X 0,Y 541.248,Z 401.786,A -85,B 0,C 180,E1 23554.475,E2 23554.475} C_VEL
LIN {X 0,Y 546.539,Z 408.356,A -85,B 0,C 180,E1 23553.135,E2 23553.135} C_VEL
LIN {X 0,Y 553.314,Z 416.958,A -85,B 0,C 180,E1 23551.535,E2 23551.535} C_VEL
LIN {X 0,Y 562.606,Z 429.371,A -85,B 0,C 180,E1 23549.509,E2 23549.509} C_VEL
LIN {X 0,Y 573.617,Z 444.659,A -85,B 0,C 180,E1 23547.321,E2 23547.321} C_VEL
LIN {X 0,Y 575.795,Z 448.147,A -85,B 0,C 180,E1 23546.902,E2 23546.902} C_VEL
LIN {X 0,Y 566.004,Z 661.624,A -85,B 0,C 180,E1 23543.683,E2 23543.683} C_VEL
LIN {X 0,Y 559.781,Z 800.774,A -85,B 0,C 180,E1 23541.592,E2 23541.592} C_VEL
LIN {X 0,Y 557.769,Z 825.938,A -85,B 0,C 180,E1 23541.112,E2 23541.112} C_VEL
LIN {X 0,Y 554.675,Z 853.503,A -85,B 0,C 180,E1 23540.393,E2 23540.393} C_VEL
LIN {X 0,Y 551.68,Z 875.247,A -85,B 0,C 180,E1 23539.681,E2 23539.681} C_VEL
LIN {X 0,Y 548.57,Z 895.002,A -85,B 0,C 180,E1 23538.909,E2 23538.909} C_VEL
LIN {X 0,Y 544.98,Z 915.222,A -85,B 0,C 180,E1 23537.991,E2 23537.991} C_VEL
LIN {X 0,Y 540.527,Z 937.986,A -85,B 0,C 180,E1 23536.787,E2 23536.787} C_VEL
LIN {X 0,Y 535,Z 963.2,A -85,B 0,C 180,E1 23535.203,E2 23535.203} C_VEL
LIN {X 0,Y 530.368,Z 982.768,A -85,B 0,C 180,E1 23533.778,E2 23533.778} C_VEL
LIN {X 0,Y 525.92,Z 1000.719,A -85,B 0,C 180,E1 23532.3,E2 23532.3} C_VEL
LIN {X 0,Y 525.705,Z 1001.573,A -85,B 0,C 180,E1 23532.226,E2 23532.226} C_VEL
LIN {X 0,Y 523.433,Z 1007.72,A -85,B 0,C 180,E1 23531.764,E2 23531.764} C_VEL
LIN {X 0,Y 514.264,Z 1024.108,A -85,B 0,C 180,E1 23530.662,E2 23530.662} C_VEL
LIN {X 0,Y 512.332,Z 1028.898,A -85,B 0,C 180,E1 23530.207,E2 23530.207} C_VEL
LIN {X 0,Y 508.001,Z 1044.432,A -85,B 0,C 180,E1 23528.459,E2 23528.459} C_VEL
LIN {X 0,Y 503.718,Z 1059.656,A -85,B 0,C 180,E1 23526.547,E2 23526.547} C_VEL
LIN {X 0,Y 499.029,Z 1076.589,A -85,B 0,C 180,E1 23524.155,E2 23524.155} C_VEL
LIN {X 0,Y 494.371,Z 1093.456,A -85,B 0,C 180,E1 23521.403,E2 23521.403} C_VEL
LIN {X 0,Y 491.159,Z 1105.801,A -85,B 0,C 180,E1 23519.113,E2 23519.113} C_VEL
LIN {X 0,Y 488.382,Z 1117.067,A -85,B 0,C 180,E1 23516.769,E2 23516.769} C_VEL
LIN {X 0,Y 486,Z 1127.613,A -85,B 0,C 180,E1 23514.297,E2 23514.297} C_VEL
LIN {X 0,Y 483.717,Z 1139.122,A -85,B 0,C 180,E1 23511.206,E2 23511.206} C_VEL
LIN {X 0,Y 482.003,Z 1149.018,A -85,B 0,C 180,E1 23508.004,E2 23508.004} C_VEL
LIN {X 0,Y 481.118,Z 1155.934,A -85,B 0,C 180,E1 23505.427,E2 23505.427} C_VEL
LIN {X 0,Y 480.513,Z 1161.725,A -85,B 0,C 180,E1 23502.865,E2 23502.865} C_VEL
LIN {X 0,Y 480.154,Z 1166.843,A -85,B 0,C 180,E1 23500.074,E2 23500.074} C_VEL
LIN {X 0,Y 479.965,Z 1171.235,A -85,B 0,C 180,E1 23496.819,E2 23496.819} C_VEL
LIN {X 0,Y 479.915,Z 1173.654,A -85,B 0,C 180,E1 23493.942,E2 23493.942} C_VEL
LIN {X 0,Y 479.909,Z 1174.726,A -85,B 0,C 180,E1 23491.433,E2 23491.433} C_VEL
LIN {X 0,Y 479.905,Z 1174.834,A -85,B 0,C 180,E1 23489.045,E2 23489.045} C_VEL
LIN {X 0,Y 479.913,Z 1173.979,A -85,B 0,C 180,E1 23486.536,E2 23486.536} C_VEL
LIN {X 0,Y 479.946,Z 1172.117,A -85,B 0,C 180,E1 23484.021,E2 23484.021} C_VEL
LIN {X 0,Y 480.038,Z 1169.246,A -85,B 0,C 180,E1 23481.496,E2 23481.496} C_VEL
LIN {X 0,Y 480.234,Z 1165.344,A -85,B 0,C 180,E1 23478.957,E2 23478.957} C_VEL
LIN {X 0,Y 480.676,Z 1160.116,A -85,B 0,C 180,E1 23476.276,E2 23476.276} C_VEL
LIN {X 0,Y 481.645,Z 1151.748,A -85,B 0,C 180,E1 23472.856,E2 23472.856} C_VEL
LIN {X 0,Y 482.975,Z 1142.96,A -85,B 0,C 180,E1 23469.9,E2 23469.9} C_VEL
LIN {X 0,Y 484.558,Z 1134.536,A -85,B 0,C 180,E1 23467.431,E2 23467.431} C_VEL
LIN {X 0,Y 486.691,Z 1124.432,A -85,B 0,C 180,E1 23464.833,E2 23464.833} C_VEL
LIN {X 0,Y 489.974,Z 1110.578,A -85,B 0,C 180,E1 23461.743,E2 23461.743} C_VEL
LIN {X 0,Y 493.42,Z 1097.099,A -85,B 0,C 180,E1 23459.158,E2 23459.158} C_VEL
LIN {X 0,Y 496.875,Z 1084.183,A -85,B 0,C 180,E1 23456.953,E2 23456.953} C_VEL
LIN {X 0,Y 500.621,Z 1070.655,A -85,B 0,C 180,E1 23454.886,E2 23454.886} C_VEL
LIN {X 0,Y 505.366,Z 1053.854,A -85,B 0,C 180,E1 23452.599,E2 23452.599} C_VEL
LIN {X 0,Y 511.003,Z 1033.724,A -85,B 0,C 180,E1 23450.221,E2 23450.221} C_VEL
LIN {X 0,Y 515.683,Z 1016.687,A -85,B 0,C 180,E1 23448.456,E2 23448.456} C_VEL
LIN {X 0,Y 520.187,Z 999.798,A -85,B 0,C 180,E1 23446.894,E2 23446.894} C_VEL
LIN {X 0,Y 524.819,Z 981.753,A -85,B 0,C 180,E1 23445.409,E2 23445.409} C_VEL
LIN {X 0,Y 530.164,Z 959.931,A -85,B 0,C 180,E1 23443.832,E2 23443.832} C_VEL
LIN {X 0,Y 535.582,Z 935.448,A -85,B 0,C 180,E1 23442.33,E2 23442.33} C_VEL
LIN {X 0,Y 539.786,Z 914.565,A -85,B 0,C 180,E1 23441.233,E2 23441.233} C_VEL
LIN {X 0,Y 543.274,Z 895.489,A -85,B 0,C 180,E1 23440.365,E2 23440.365} C_VEL
LIN {X 0,Y 546.658,Z 874.695,A -85,B 0,C 180,E1 23439.554,E2 23439.554} C_VEL
LIN {X 0,Y 550.006,Z 850.907,A -85,B 0,C 180,E1 23438.782,E2 23438.782} C_VEL
LIN {X 0,Y 553.102,Z 822.698,A -85,B 0,C 180,E1 23438.075,E2 23438.075} C_VEL
LIN {X 0,Y 554.949,Z 799.825,A -85,B 0,C 180,E1 23437.648,E2 23437.648} C_VEL
LIN {X 0,Y 564.622,Z 591.381,A -85,B 0,C 180,E1 23434.503,E2 23434.503} C_VEL
LIN {X 0,Y 571.273,Z 452.334,A -85,B 0,C 180,E1 23432.384,E2 23432.384} C_VEL
LIN {X 0,Y 560.597,Z 437.161,A -85,B 0,C 180,E1 23430.227,E2 23430.227} C_VEL
LIN {X 0,Y 552.094,Z 425.771,A -85,B 0,C 180,E1 23428.357,E2 23428.357} C_VEL
LIN {X 0,Y 544.578,Z 415.951,A -85,B 0,C 180,E1 23426.557,E2 23426.557} C_VEL
LIN {X 0,Y 540.459,Z 410.844,A -85,B 0,C 180,E1 23425.506,E2 23425.506} C_VEL
LIN {X 0,Y 536.691,Z 406.091,A -85,B 0,C 180,E1 23424.49,E2 23424.49} C_VEL
LIN {X 0,Y 532.462,Z 400.826,A -85,B 0,C 180,E1 23423.284,E2 23423.284} C_VEL
LIN {X 0,Y 528.105,Z 395.541,A -85,B 0,C 180,E1 23421.959,E2 23421.959} C_VEL
LIN {X 0,Y 524.229,Z 390.84,A -85,B 0,C 180,E1 23420.692,E2 23420.692} C_VEL
LIN {X 0,Y 519.474,Z 385.435,A -85,B 0,C 180,E1 23419.013,E2 23419.013} C_VEL
LIN {X 0,Y 518.302,Z 383.868,A -85,B 0,C 180,E1 23418.561,E2 23418.561} C_VEL
LIN {X 0,Y 514.888,Z 380.59,A -85,B 0,C 180,E1 23417.227,E2 23417.227} C_VEL
LIN {X 0,Y 513.074,Z 377.779,A -85,B 0,C 180,E1 23416.414,E2 23416.414} C_VEL
LIN {X 0,Y 509.682,Z 374.937,A -85,B 0,C 180,E1 23414.892,E2 23414.892} C_VEL
LIN {X 0,Y 507.658,Z 371.422,A -85,B 0,C 180,E1 23413.788,E2 23413.788} C_VEL
LIN {X 0,Y 503.858,Z 368.751,A -85,B 0,C 180,E1 23411.678,E2 23411.678} C_VEL
LIN {X 0,Y 502.091,Z 365.493,A -85,B 0,C 180,E1 23410.383,E2 23410.383} C_VEL
LIN {X 0,Y 501.742,Z 364.777,A -85,B 0,C 180,E1 23410.1,E2 23410.1} C_VEL
LIN {X 0,Y 497.868,Z 362.421,A -85,B 0,C 180,E1 23406.805,E2 23406.805} C_VEL
LIN {X 0,Y 496.03,Z 359.063,A -85,B 0,C 180,E1 23403.93,E2 23403.93} C_VEL
LIN {X 0,Y 495.708,Z 357.983,A -85,B 0,C 180,E1 23403.006,E2 23403.006} C_VEL
LIN {X 0,Y 495.881,Z 358.113,A -85,B 0,C 180,E1 23396.995,E2 23396.995} C_VEL
LIN {X 0,Y 496.86,Z 361.016,A -85,B 0,C 180,E1 23394.92,E2 23394.92} C_VEL
LIN {X 0,Y 499.717,Z 363.929,A -85,B 0,C 180,E1 23391.833,E2 23391.833} C_VEL
LIN {X 0,Y 501.91,Z 364.952,A -85,B 0,C 180,E1 23390.193,E2 23390.193} C_VEL
LIN {X 0,Y 503.712,Z 368.466,A -85,B 0,C 180,E1 23388.84,E2 23388.84} C_VEL
LIN {X 0,Y 506.48,Z 370.889,A -85,B 0,C 180,E1 23387.226,E2 23387.226} C_VEL
LIN {X 0,Y 507.823,Z 371.701,A -85,B 0,C 180,E1 23386.536,E2 23386.536} C_VEL
LIN {X 0,Y 510.159,Z 375.413,A -85,B 0,C 180,E1 23385.297,E2 23385.297} C_VEL
LIN {X 0,Y 513.593,Z 378.349,A -85,B 0,C 180,E1 23383.777,E2 23383.777} C_VEL
LIN {X 0,Y 516.486,Z 382.423,A -85,B 0,C 180,E1 23382.538,E2 23382.538} C_VEL
LIN {X 0,Y 518.719,Z 384.578,A -85,B 0,C 180,E1 23381.687,E2 23381.687} C_VEL
LIN {X 0,Y 523.336,Z 390.512,A -85,B 0,C 180,E1 23380.001,E2 23380.001} C_VEL
LIN {X 0,Y 527.379,Z 395.659,A -85,B 0,C 180,E1 23378.652,E2 23378.652} C_VEL
LIN {X 0,Y 532.167,Z 401.934,A -85,B 0,C 180,E1 23377.17,E2 23377.17} C_VEL
LIN {X 0,Y 539.154,Z 411.326,A -85,B 0,C 180,E1 23375.191,E2 23375.191} C_VEL
LIN {X 0,Y 548.74,Z 424.629,A -85,B 0,C 180,E1 23372.754,E2 23372.754} C_VEL
LIN {X 0,Y 560.258,Z 441.667,A -85,B 0,C 180,E1 23370.137,E2 23370.137} C_VEL
LIN {X 0,Y 571.421,Z 459.345,A -85,B 0,C 180,E1 23367.848,E2 23367.848} C_VEL
LIN {X 0,Y 561.392,Z 671.95,A -85,B 0,C 180,E1 23364.627,E2 23364.627} C_VEL
LIN {X 0,Y 554.479,Z 823.103,A -85,B 0,C 180,E1 23362.345,E2 23362.345} C_VEL
LIN {X 0,Y 552.279,Z 849.224,A -85,B 0,C 180,E1 23361.856,E2 23361.856} C_VEL
LIN {X 0,Y 548.98,Z 876.705,A -85,B 0,C 180,E1 23361.154,E2 23361.154} C_VEL
LIN {X 0,Y 545.853,Z 898.353,A -85,B 0,C 180,E1 23360.458,E2 23360.458} C_VEL
LIN {X 0,Y 542.425,Z 919.143,A -85,B 0,C 180,E1 23359.659,E2 23359.659} C_VEL
LIN {X 0,Y 538.679,Z 939.539,A -85,B 0,C 180,E1 23358.74,E2 23358.74} C_VEL
LIN {X 0,Y 533.639,Z 964.588,A -85,B 0,C 180,E1 23357.421,E2 23357.421} C_VEL
LIN {X 0,Y 528.221,Z 988.452,A -85,B 0,C 180,E1 23355.918,E2 23355.918} C_VEL
LIN {X 0,Y 523.523,Z 1008.054,A -85,B 0,C 180,E1 23354.501,E2 23354.501} C_VEL
LIN {X 0,Y 518.935,Z 1026.362,A -85,B 0,C 180,E1 23353.005,E2 23353.005} C_VEL
LIN {X 0,Y 513.652,Z 1046.819,A -85,B 0,C 180,E1 23351.119,E2 23351.119} C_VEL
LIN {X 0,Y 507.958,Z 1068.011,A -85,B 0,C 180,E1 23348.858,E2 23348.858} C_VEL
LIN {X 0,Y 503.518,Z 1084.599,A -85,B 0,C 180,E1 23346.848,E2 23346.848} C_VEL
LIN {X 0,Y 499.475,Z 1099.83,A -85,B 0,C 180,E1 23344.786,E2 23344.786} C_VEL
LIN {X 0,Y 495.147,Z 1116.794,A -85,B 0,C 180,E1 23342.207,E2 23342.207} C_VEL
LIN {X 0,Y 491.12,Z 1132.881,A -85,B 0,C 180,E1 23339.38,E2 23339.38} C_VEL
LIN {X 0,Y 488.282,Z 1145.282,A -85,B 0,C 180,E1 23336.907,E2 23336.907} C_VEL
LIN {X 0,Y 485.941,Z 1156.327,A -85,B 0,C 180,E1 23334.429,E2 23334.429} C_VEL
LIN {X 0,Y 483.778,Z 1167.973,A -85,B 0,C 180,E1 23331.458,E2 23331.458} C_VEL
LIN {X 0,Y 482.151,Z 1178.088,A -85,B 0,C 180,E1 23328.373,E2 23328.373} C_VEL
LIN {X 0,Y 481.173,Z 1185.439,A -85,B 0,C 180,E1 23325.672,E2 23325.672} C_VEL
LIN {X 0,Y 480.556,Z 1191.31,A -85,B 0,C 180,E1 23323.108,E2 23323.108} C_VEL
LIN {X 0,Y 480.196,Z 1196.094,A -85,B 0,C 180,E1 23320.558,E2 23320.558} C_VEL
LIN {X 0,Y 480.008,Z 1199.985,A -85,B 0,C 180,E1 23317.902,E2 23317.902} C_VEL
LIN {X 0,Y 479.923,Z 1203.193,A -85,B 0,C 180,E1 23314.78,E2 23314.78} C_VEL
LIN {X 0,Y 479.908,Z 1204.689,A -85,B 0,C 180,E1 23311.671,E2 23311.671} C_VEL
LIN {X 0,Y 479.902,Z 1204.848,A -85,B 0,C 180,E1 23309.164,E2 23309.164} C_VEL
LIN {X 0,Y 479.915,Z 1204.02,A -85,B 0,C 180,E1 23306.656,E2 23306.656} C_VEL
LIN {X 0,Y 479.942,Z 1202.187,A -85,B 0,C 180,E1 23304.141,E2 23304.141} C_VEL
LIN {X 0,Y 480.03,Z 1199.345,A -85,B 0,C 180,E1 23301.616,E2 23301.616} C_VEL
LIN {X 0,Y 480.227,Z 1195.474,A -85,B 0,C 180,E1 23299.078,E2 23299.078} C_VEL
LIN {X 0,Y 480.66,Z 1190.292,A -85,B 0,C 180,E1 23296.405,E2 23296.405} C_VEL
LIN {X 0,Y 481.54,Z 1182.564,A -85,B 0,C 180,E1 23293.185,E2 23293.185} C_VEL
LIN {X 0,Y 482.802,Z 1173.837,A -85,B 0,C 180,E1 23290.271,E2 23290.271} C_VEL
LIN {X 0,Y 484.375,Z 1164.552,A -85,B 0,C 180,E1 23287.639,E2 23287.639} C_VEL
LIN {X 0,Y 486.258,Z 1154.756,A -85,B 0,C 180,E1 23285.199,E2 23285.199} C_VEL
LIN {X 0,Y 488.677,Z 1143.533,A -85,B 0,C 180,E1 23282.722,E2 23282.722} C_VEL
LIN {X 0,Y 492.283,Z 1128.239,A -85,B 0,C 180,E1 23279.755,E2 23279.755} C_VEL
LIN {X 0,Y 496.105,Z 1112.831,A -85,B 0,C 180,E1 23277.17,E2 23277.17} C_VEL
LIN {X 0,Y 499.693,Z 1098.972,A -85,B 0,C 180,E1 23275.091,E2 23275.091} C_VEL
LIN {X 0,Y 503.767,Z 1083.66,A -85,B 0,C 180,E1 23273.031,E2 23273.031} C_VEL
LIN {X 0,Y 508.756,Z 1065.168,A -85,B 0,C 180,E1 23270.814,E2 23270.814} C_VEL
LIN {X 0,Y 514.476,Z 1043.59,A -85,B 0,C 180,E1 23268.575,E2 23268.575} C_VEL
LIN {X 0,Y 519.105,Z 1025.665,A -85,B 0,C 180,E1 23266.937,E2 23266.937} C_VEL
LIN {X 0,Y 523.706,Z 1007.281,A -85,B 0,C 180,E1 23265.442,E2 23265.442} C_VEL
LIN {X 0,Y 528.416,Z 987.6,A -85,B 0,C 180,E1 23264.026,E2 23264.026} C_VEL
LIN {X 0,Y 534.045,Z 962.541,A -85,B 0,C 180,E1 23262.468,E2 23262.468} C_VEL
LIN {X 0,Y 538.673,Z 939.487,A -85,B 0,C 180,E1 23261.259,E2 23261.259} C_VEL
LIN {X 0,Y 542.417,Z 919.073,A -85,B 0,C 180,E1 23260.34,E2 23260.34} C_VEL
LIN {X 0,Y 545.846,Z 898.266,A -85,B 0,C 180,E1 23259.541,E2 23259.541} C_VEL
LIN {X 0,Y 549.096,Z 875.728,A -85,B 0,C 180,E1 23258.82,E2 23258.82} C_VEL
LIN {X 0,Y 552.447,Z 847.102,A -85,B 0,C 180,E1 23258.104,E2 23258.104} C_VEL
LIN {X 0,Y 554.48,Z 822.641,A -85,B 0,C 180,E1 23257.65,E2 23257.65} C_VEL
LIN {X 0,Y 563.771,Z 619.291,A -85,B 0,C 180,E1 23254.583,E2 23254.583} C_VEL
LIN {X 0,Y 571.315,Z 459.234,A -85,B 0,C 180,E1 23252.144,E2 23252.144} C_VEL
LIN {X 0,Y 560.087,Z 441.471,A -85,B 0,C 180,E1 23249.844,E2 23249.844} C_VEL
LIN {X 0,Y 548.561,Z 424.426,A -85,B 0,C 180,E1 23247.227,E2 23247.227} C_VEL
LIN {X 0,Y 537.615,Z 409.116,A -85,B 0,C 180,E1 23244.416,E2 23244.416} C_VEL
LIN {X 0,Y 529.875,Z 398.921,A -85,B 0,C 180,E1 23242.173,E2 23242.173} C_VEL
LIN {X 0,Y 525.362,Z 393.108,A -85,B 0,C 180,E1 23240.732,E2 23240.732} C_VEL
LIN {X 0,Y 520.846,Z 387.364,A -85,B 0,C 180,E1 23239.164,E2 23239.164} C_VEL
LIN {X 0,Y 517.743,Z 383.508,A -85,B 0,C 180,E1 23237.999,E2 23237.999} C_VEL
LIN {X 0,Y 514.523,Z 380.009,A -85,B 0,C 180,E1 23236.715,E2 23236.715} C_VEL
LIN {X 0,Y 513.069,Z 377.765,A -85,B 0,C 180,E1 23236.066,E2 23236.066} C_VEL
LIN {X 0,Y 509.55,Z 374.698,A -85,B 0,C 180,E1 23234.489,E2 23234.489} C_VEL
LIN {X 0,Y 507.613,Z 371.374,A -85,B 0,C 180,E1 23233.441,E2 23233.441} C_VEL
LIN {X 0,Y 504.231,Z 369.144,A -85,B 0,C 180,E1 23231.612,E2 23231.612} C_VEL
LIN {X 0,Y 502.073,Z 365.474,A -85,B 0,C 180,E1 23230.093,E2 23230.093} C_VEL
LIN {X 0,Y 501.635,Z 364.717,A -85,B 0,C 180,E1 23229.755,E2 23229.755} C_VEL
LIN {X 0,Y 497.71,Z 362.313,A -85,B 0,C 180,E1 23226.46,E2 23226.46} C_VEL
LIN {X 0,Y 495.882,Z 358.458,A -85,B 0,C 180,E1 23223.584,E2 23223.584} C_VEL
LIN {X 0,Y 495.69,Z 357.978,A -85,B 0,C 180,E1 23223.122,E2 23223.122} C_VEL
LIN {X 0,Y 495.828,Z 358.167,A -85,B 0,C 180,E1 23216.068,E2 23216.068} C_VEL
LIN {X 0,Y 497.104,Z 361.505,A -85,B 0,C 180,E1 23213.764,E2 23213.764} C_VEL
LIN {X 0,Y 500.609,Z 364.377,A -85,B 0,C 180,E1 23210.457,E2 23210.457} C_VEL
LIN {X 0,Y 501.921,Z 365.081,A -85,B 0,C 180,E1 23209.526,E2 23209.526} C_VEL
LIN {X 0,Y 503.545,Z 368.362,A -85,B 0,C 180,E1 23208.314,E2 23208.314} C_VEL
LIN {X 0,Y 507.082,Z 371.187,A -85,B 0,C 180,E1 23206.313,E2 23206.313} C_VEL
LIN {X 0,Y 507.837,Z 371.767,A -85,B 0,C 180,E1 23205.927,E2 23205.927} C_VEL
LIN {X 0,Y 510.135,Z 375.494,A -85,B 0,C 180,E1 23204.715,E2 23204.715} C_VEL
LIN {X 0,Y 513.472,Z 378.294,A -85,B 0,C 180,E1 23203.25,E2 23203.25} C_VEL
LIN {X 0,Y 516.249,Z 382.181,A -85,B 0,C 180,E1 23202.064,E2 23202.064} C_VEL
LIN {X 0,Y 519.003,Z 384.675,A -85,B 0,C 180,E1 23201.028,E2 23201.028} C_VEL
LIN {X 0,Y 522.547,Z 389.148,A -85,B 0,C 180,E1 23199.736,E2 23199.736} C_VEL
LIN {X 0,Y 524.329,Z 391.012,A -85,B 0,C 180,E1 23199.137,E2 23199.137} C_VEL
LIN {X 0,Y 528.233,Z 395.678,A -85,B 0,C 180,E1 23197.871,E2 23197.871} C_VEL
LIN {X 0,Y 534.272,Z 403.052,A -85,B 0,C 180,E1 23196.068,E2 23196.068} C_VEL
LIN {X 0,Y 539.153,Z 409.184,A -85,B 0,C 180,E1 23194.722,E2 23194.722} C_VEL
LIN {X 0,Y 546.668,Z 418.499,A -85,B 0,C 180,E1 23192.818,E2 23192.818} C_VEL
LIN {X 0,Y 558.04,Z 433.665,A -85,B 0,C 180,E1 23190.213,E2 23190.213} C_VEL
LIN {X 0,Y 569.73,Z 450.051,A -85,B 0,C 180,E1 23187.815,E2 23187.815} C_VEL
LIN {X 0,Y 571.251,Z 452.677,A -85,B 0,C 180,E1 23187.51,E2 23187.51} C_VEL
LIN {X 0,Y 561.071,Z 666.889,A -85,B 0,C 180,E1 23184.267,E2 23184.267} C_VEL
LIN {X 0,Y 554.841,Z 801.091,A -85,B 0,C 180,E1 23182.239,E2 23182.239} C_VEL
LIN {X 0,Y 552.737,Z 826.63,A -85,B 0,C 180,E1 23181.75,E2 23181.75} C_VEL
LIN {X 0,Y 549.556,Z 853.996,A -85,B 0,C 180,E1 23181.033,E2 23181.033} C_VEL
LIN {X 0,Y 546.645,Z 874.61,A -85,B 0,C 180,E1 23180.358,E2 23180.358} C_VEL
LIN {X 0,Y 543.292,Z 895.277,A -85,B 0,C 180,E1 23179.552,E2 23179.552} C_VEL
LIN {X 0,Y 539.587,Z 915.496,A -85,B 0,C 180,E1 23178.631,E2 23178.631} C_VEL
LIN {X 0,Y 534.987,Z 938.261,A -85,B 0,C 180,E1 23177.422,E2 23177.422} C_VEL
LIN {X 0,Y 529.387,Z 962.984,A -85,B 0,C 180,E1 23175.865,E2 23175.865} C_VEL
LIN {X 0,Y 524.656,Z 982.317,A -85,B 0,C 180,E1 23174.456,E2 23174.456} C_VEL
LIN {X 0,Y 520.033,Z 1000.334,A -85,B 0,C 180,E1 23172.968,E2 23172.968} C_VEL
LIN {X 0,Y 515.209,Z 1018.405,A -85,B 0,C 180,E1 23171.287,E2 23171.287} C_VEL
LIN {X 0,Y 512.332,Z 1028.898,A -85,B 0,C 180,E1 23170.207,E2 23170.207} C_VEL
LIN {X 0,Y 509.993,Z 1034.613,A -85,B 0,C 180,E1 23169.67,E2 23169.67} C_VEL
LIN {X 0,Y 500.68,Z 1049.862,A -85,B 0,C 180,E1 23168.376,E2 23168.376} C_VEL
LIN {X 0,Y 498.709,Z 1054.35,A -85,B 0,C 180,E1 23167.861,E2 23167.861} C_VEL
LIN {X 0,Y 493.973,Z 1070.396,A -85,B 0,C 180,E1 23165.658,E2 23165.658} C_VEL
LIN {X 0,Y 489.814,Z 1084.722,A -85,B 0,C 180,E1 23163.446,E2 23163.446} C_VEL
LIN {X 0,Y 486.024,Z 1098.294,A -85,B 0,C 180,E1 23161.088,E2 23161.088} C_VEL
LIN {X 0,Y 481.823,Z 1113.976,A -85,B 0,C 180,E1 23157.968,E2 23157.968} C_VEL
LIN {X 0,Y 479.01,Z 1125.387,A -85,B 0,C 180,E1 23155.331,E2 23155.331} C_VEL
LIN {X 0,Y 476.877,Z 1134.948,A -85,B 0,C 180,E1 23152.823,E2 23152.823} C_VEL
LIN {X 0,Y 475.207,Z 1143.346,A -85,B 0,C 180,E1 23150.314,E2 23150.314} C_VEL
LIN {X 0,Y 473.863,Z 1151.326,A -85,B 0,C 180,E1 23147.562,E2 23147.562} C_VEL
LIN {X 0,Y 472.776,Z 1159.689,A -85,B 0,C 180,E1 23144.076,E2 23144.076} C_VEL
LIN {X 0,Y 472.269,Z 1165.189,A -85,B 0,C 180,E1 23141.232,E2 23141.232} C_VEL
LIN {X 0,Y 472.056,Z 1169.124,A -85,B 0,C 180,E1 23138.649,E2 23138.649} C_VEL
LIN {X 0,Y 471.952,Z 1172.029,A -85,B 0,C 180,E1 23136.081,E2 23136.081} C_VEL
LIN {X 0,Y 471.914,Z 1173.924,A -85,B 0,C 180,E1 23133.523,E2 23133.523} C_VEL
LIN {X 0,Y 471.906,Z 1174.817,A -85,B 0,C 180,E1 23130.971,E2 23130.971} C_VEL
LIN {X 0,Y 471.907,Z 1174.72,A -85,B 0,C 180,E1 23128.422,E2 23128.422} C_VEL
LIN {X 0,Y 471.92,Z 1173.567,A -85,B 0,C 180,E1 23125.747,E2 23125.747} C_VEL
LIN {X 0,Y 471.989,Z 1170.68,A -85,B 0,C 180,E1 23122.453,E2 23122.453} C_VEL
LIN {X 0,Y 472.204,Z 1166.373,A -85,B 0,C 180,E1 23119.385,E2 23119.385} C_VEL
LIN {X 0,Y 472.594,Z 1161.501,A -85,B 0,C 180,E1 23116.718,E2 23116.718} C_VEL
LIN {X 0,Y 473.324,Z 1155.029,A -85,B 0,C 180,E1 23113.809,E2 23113.809} C_VEL
LIN {X 0,Y 474.697,Z 1146.392,A -85,B 0,C 180,E1 23110.561,E2 23110.561} C_VEL
LIN {X 0,Y 476.627,Z 1136.151,A -85,B 0,C 180,E1 23107.425,E2 23107.425} C_VEL
LIN {X 0,Y 478.69,Z 1126.716,A -85,B 0,C 180,E1 23104.912,E2 23104.912} C_VEL
LIN {X 0,Y 481.291,Z 1116.031,A -85,B 0,C 180,E1 23102.402,E2 23102.402} C_VEL
LIN {X 0,Y 485.011,Z 1102.066,A -85,B 0,C 180,E1 23099.513,E2 23099.513} C_VEL
LIN {X 0,Y 489.47,Z 1085.967,A -85,B 0,C 180,E1 23096.668,E2 23096.668} C_VEL
LIN {X 0,Y 493.363,Z 1072.494,A -85,B 0,C 180,E1 23094.561,E2 23094.561} C_VEL
LIN {X 0,Y 497.678,Z 1057.771,A -85,B 0,C 180,E1 23092.502,E2 23092.502} C_VEL
LIN {X 0,Y 502.868,Z 1040.135,A -85,B 0,C 180,E1 23090.31,E2 23090.31} C_VEL
LIN {X 0,Y 509.007,Z 1018.817,A -85,B 0,C 180,E1 23088.021,E2 23088.021} C_VEL
LIN {X 0,Y 513.877,Z 1001.264,A -85,B 0,C 180,E1 23086.372,E2 23086.372} C_VEL
LIN {X 0,Y 518.646,Z 983.374,A -85,B 0,C 180,E1 23084.879,E2 23084.879} C_VEL
LIN {X 0,Y 523.502,Z 964.215,A -85,B 0,C 180,E1 23083.467,E2 23083.467} C_VEL
LIN {X 0,Y 529.293,Z 939.695,A -85,B 0,C 180,E1 23081.903,E2 23081.903} C_VEL
LIN {X 0,Y 534.213,Z 916.159,A -85,B 0,C 180,E1 23080.644,E2 23080.644} C_VEL
LIN {X 0,Y 538.072,Z 895.745,A -85,B 0,C 180,E1 23079.709,E2 23079.709} C_VEL
LIN {X 0,Y 541.563,Z 874.949,A -85,B 0,C 180,E1 23078.896,E2 23078.896} C_VEL
LIN {X 0,Y 544.978,Z 851.374,A -85,B 0,C 180,E1 23078.13,E2 23078.13} C_VEL
LIN {X 0,Y 548.18,Z 823.104,A -85,B 0,C 180,E1 23077.419,E2 23077.419} C_VEL
LIN {X 0,Y 550.086,Z 800.18,A -85,B 0,C 180,E1 23076.989,E2 23076.989} C_VEL
LIN {X 0,Y 560.08,Z 592.474,A -85,B 0,C 180,E1 23073.84,E2 23073.84} C_VEL
LIN {X 0,Y 566.847,Z 456.812,A -85,B 0,C 180,E1 23071.772,E2 23071.772} C_VEL
LIN {X 0,Y 556.26,Z 441.841,A -85,B 0,C 180,E1 23069.566,E2 23069.566} C_VEL
LIN {X 0,Y 547.06,Z 429.324,A -85,B 0,C 180,E1 23067.455,E2 23067.455} C_VEL
LIN {X 0,Y 539.118,Z 419.097,A -85,B 0,C 180,E1 23065.456,E2 23065.456} C_VEL
LIN {X 0,Y 534.279,Z 413.043,A -85,B 0,C 180,E1 23064.137,E2 23064.137} C_VEL
LIN {X 0,Y 530.288,Z 408.014,A -85,B 0,C 180,E1 23062.974,E2 23062.974} C_VEL
LIN {X 0,Y 526.157,Z 402.932,A -85,B 0,C 180,E1 23061.692,E2 23061.692} C_VEL
LIN {X 0,Y 522.192,Z 397.982,A -85,B 0,C 180,E1 23060.366,E2 23060.366} C_VEL
LIN {X 0,Y 517.861,Z 393.114,A -85,B 0,C 180,E1 23058.811,E2 23058.811} C_VEL
LIN {X 0,Y 516.634,Z 391.47,A -85,B 0,C 180,E1 23058.331,E2 23058.331} C_VEL
LIN {X 0,Y 513.152,Z 387.96,A -85,B 0,C 180,E1 23056.936,E2 23056.936} C_VEL
LIN {X 0,Y 511.607,Z 385.517,A -85,B 0,C 180,E1 23056.229,E2 23056.229} C_VEL
LIN {X 0,Y 508.265,Z 382.628,A -85,B 0,C 180,E1 23054.701,E2 23054.701} C_VEL
LIN {X 0,Y 506.262,Z 379.219,A -85,B 0,C 180,E1 23053.593,E2 23053.593} C_VEL
LIN {X 0,Y 502.537,Z 376.448,A -85,B 0,C 180,E1 23051.477,E2 23051.477} C_VEL
LIN {X 0,Y 500.742,Z 373.046,A -85,B 0,C 180,E1 23050.121,E2 23050.121} C_VEL
LIN {X 0,Y 500.132,Z 372.526,A -85,B 0,C 180,E1 23049.668,E2 23049.668} C_VEL
LIN {X 0,Y 496.318,Z 369.767,A -85,B 0,C 180,E1 23046.129,E2 23046.129} C_VEL
LIN {X 0,Y 494.734,Z 365.923,A -85,B 0,C 180,E1 23043.012,E2 23043.012} C_VEL
LIN {X 0,Y 494.872,Z 366.113,A -85,B 0,C 180,E1 23037.047,E2 23037.047} C_VEL
LIN {X 0,Y 495.958,Z 369.155,A -85,B 0,C 180,E1 23034.795,E2 23034.795} C_VEL
LIN {X 0,Y 499.027,Z 372.042,A -85,B 0,C 180,E1 23031.589,E2 23031.589} C_VEL
LIN {X 0,Y 500.692,Z 372.882,A -85,B 0,C 180,E1 23030.343,E2 23030.343} C_VEL
LIN {X 0,Y 502.732,Z 376.606,A -85,B 0,C 180,E1 23028.818,E2 23028.818} C_VEL
LIN {X 0,Y 505.737,Z 378.977,A -85,B 0,C 180,E1 23027.09,E2 23027.09} C_VEL
LIN {X 0,Y 506.47,Z 379.585,A -85,B 0,C 180,E1 23026.703,E2 23026.703} C_VEL
LIN {X 0,Y 508.96,Z 383.346,A -85,B 0,C 180,E1 23025.377,E2 23025.377} C_VEL
LIN {X 0,Y 512.052,Z 386.047,A -85,B 0,C 180,E1 23023.989,E2 23023.989} C_VEL
LIN {X 0,Y 515.116,Z 390.243,A -85,B 0,C 180,E1 23022.665,E2 23022.665} C_VEL
LIN {X 0,Y 517.319,Z 392.51,A -85,B 0,C 180,E1 23021.811,E2 23021.811} C_VEL
LIN {X 0,Y 521.603,Z 398.081,A -85,B 0,C 180,E1 23020.224,E2 23020.224} C_VEL
LIN {X 0,Y 525.517,Z 403.145,A -85,B 0,C 180,E1 23018.895,E2 23018.895} C_VEL
LIN {X 0,Y 530.247,Z 409.426,A -85,B 0,C 180,E1 23017.405,E2 23017.405} C_VEL
LIN {X 0,Y 537.155,Z 418.864,A -85,B 0,C 180,E1 23015.415,E2 23015.415} C_VEL
LIN {X 0,Y 546.349,Z 431.813,A -85,B 0,C 180,E1 23013.037,E2 23013.037} C_VEL
LIN {X 0,Y 557.421,Z 448.399,A -85,B 0,C 180,E1 23010.472,E2 23010.472} C_VEL
LIN {X 0,Y 566.937,Z 463.693,A -85,B 0,C 180,E1 23008.468,E2 23008.468} C_VEL
LIN {X 0,Y 556.592,Z 675.389,A -85,B 0,C 180,E1 23005.247,E2 23005.247} C_VEL
LIN {X 0,Y 549.591,Z 822.964,A -85,B 0,C 180,E1 23003.008,E2 23003.008} C_VEL
LIN {X 0,Y 547.282,Z 849.571,A -85,B 0,C 180,E1 23002.507,E2 23002.507} C_VEL
LIN {X 0,Y 543.925,Z 876.558,A -85,B 0,C 180,E1 23001.814,E2 23001.814} C_VEL
LIN {X 0,Y 540.713,Z 898.094,A -85,B 0,C 180,E1 23001.122,E2 23001.122} C_VEL
LIN {X 0,Y 537.188,Z 918.84,A -85,B 0,C 180,E1 23000.324,E2 23000.324} C_VEL
LIN {X 0,Y 533.307,Z 939.275,A -85,B 0,C 180,E1 22999.403,E2 22999.403} C_VEL
LIN {X 0,Y 528.317,Z 963.325,A -85,B 0,C 180,E1 22998.134,E2 22998.134} C_VEL
LIN {X 0,Y 522.703,Z 987.365,A -85,B 0,C 180,E1 22996.626,E2 22996.626} C_VEL
LIN {X 0,Y 518.01,Z 1006.301,A -85,B 0,C 180,E1 22995.26,E2 22995.26} C_VEL
LIN {X 0,Y 513.394,Z 1024.066,A -85,B 0,C 180,E1 22993.816,E2 22993.816} C_VEL
LIN {X 0,Y 508.726,Z 1041.42,A -85,B 0,C 180,E1 22992.235,E2 22992.235} C_VEL
LIN {X 0,Y 503.629,Z 1059.991,A -85,B 0,C 180,E1 22990.331,E2 22990.331} C_VEL
LIN {X 0,Y 497.586,Z 1081.503,A -85,B 0,C 180,E1 22987.797,E2 22987.797} C_VEL
LIN {X 0,Y 493.26,Z 1096.976,A -85,B 0,C 180,E1 22985.717,E2 22985.717} C_VEL
LIN {X 0,Y 489.422,Z 1110.985,A -85,B 0,C 180,E1 22983.617,E2 22983.617} C_VEL
LIN {X 0,Y 485.872,Z 1124.392,A -85,B 0,C 180,E1 22981.375,E2 22981.375} C_VEL
LIN {X 0,Y 482.222,Z 1139.062,A -85,B 0,C 180,E1 22978.618,E2 22978.618} C_VEL
LIN {X 0,Y 478.887,Z 1153.421,A -85,B 0,C 180,E1 22975.474,E2 22975.474} C_VEL
LIN {X 0,Y 476.813,Z 1163.476,A -85,B 0,C 180,E1 22972.957,E2 22972.957} C_VEL
LIN {X 0,Y 475.187,Z 1172.321,A -85,B 0,C 180,E1 22970.444,E2 22970.444} C_VEL
LIN {X 0,Y 473.958,Z 1180.06,A -85,B 0,C 180,E1 22967.925,E2 22967.925} C_VEL
LIN {X 0,Y 473.052,Z 1187.25,A -85,B 0,C 180,E1 22965.194,E2 22965.194} C_VEL
LIN {X 0,Y 472.356,Z 1194.232,A -85,B 0,C 180,E1 22961.848,E2 22961.848} C_VEL
LIN {X 0,Y 472.063,Z 1198.864,A -85,B 0,C 180,E1 22958.895,E2 22958.895} C_VEL
LIN {X 0,Y 471.954,Z 1201.844,A -85,B 0,C 180,E1 22956.325,E2 22956.325} C_VEL
LIN {X 0,Y 471.914,Z 1203.814,A -85,B 0,C 180,E1 22953.766,E2 22953.766} C_VEL
LIN {X 0,Y 471.913,Z 1204.757,A -85,B 0,C 180,E1 22951.335,E2 22951.335} C_VEL
LIN {X 0,Y 471.911,Z 1204.802,A -85,B 0,C 180,E1 22948.907,E2 22948.907} C_VEL
LIN {X 0,Y 471.915,Z 1203.949,A -85,B 0,C 180,E1 22946.477,E2 22946.477} C_VEL
LIN {X 0,Y 471.945,Z 1202.184,A -85,B 0,C 180,E1 22944.041,E2 22944.041} C_VEL
LIN {X 0,Y 472.034,Z 1199.487,A -85,B 0,C 180,E1 22941.584,E2 22941.584} C_VEL
LIN {X 0,Y 472.226,Z 1195.884,A -85,B 0,C 180,E1 22939.138,E2 22939.138} C_VEL
LIN {X 0,Y 472.638,Z 1191.052,A -85,B 0,C 180,E1 22936.544,E2 22936.544} C_VEL
LIN {X 0,Y 473.223,Z 1185.696,A -85,B 0,C 180,E1 22934.183,E2 22934.183} C_VEL
LIN {X 0,Y 474.161,Z 1178.718,A -85,B 0,C 180,E1 22931.613,E2 22931.613} C_VEL
LIN {X 0,Y 475.635,Z 1169.833,A -85,B 0,C 180,E1 22928.803,E2 22928.803} C_VEL
LIN {X 0,Y 478.097,Z 1157.11,A -85,B 0,C 180,E1 22925.407,E2 22925.407} C_VEL
LIN {X 0,Y 480.656,Z 1145.598,A -85,B 0,C 180,E1 22922.765,E2 22922.765} C_VEL
LIN {X 0,Y 483.453,Z 1133.888,A -85,B 0,C 180,E1 22920.377,E2 22920.377} C_VEL
LIN {X 0,Y 487.008,Z 1120.113,A -85,B 0,C 180,E1 22917.877,E2 22917.877} C_VEL
LIN {X 0,Y 492.091,Z 1101.271,A -85,B 0,C 180,E1 22914.899,E2 22914.899} C_VEL
LIN {X 0,Y 496.491,Z 1085.362,A -85,B 0,C 180,E1 22912.703,E2 22912.703} C_VEL
LIN {X 0,Y 500.914,Z 1069.516,A -85,B 0,C 180,E1 22910.747,E2 22910.747} C_VEL
LIN {X 0,Y 506.095,Z 1050.983,A -85,B 0,C 180,E1 22908.711,E2 22908.711} C_VEL
LIN {X 0,Y 512.218,Z 1028.488,A -85,B 0,C 180,E1 22906.567,E2 22906.567} C_VEL
LIN {X 0,Y 517.236,Z 1009.232,A -85,B 0,C 180,E1 22904.968,E2 22904.968} C_VEL
LIN {X 0,Y 521.985,Z 990.159,A -85,B 0,C 180,E1 22903.567,E2 22903.567} C_VEL
LIN {X 0,Y 526.787,Z 969.74,A -85,B 0,C 180,E1 22902.249,E2 22902.249} C_VEL
LIN {X 0,Y 532.466,Z 943.542,A -85,B 0,C 180,E1 22900.806,E2 22900.806} C_VEL
LIN {X 0,Y 536.938,Z 920.092,A -85,B 0,C 180,E1 22899.73,E2 22899.73} C_VEL
LIN {X 0,Y 540.467,Z 899.479,A -85,B 0,C 180,E1 22898.93,E2 22898.93} C_VEL
LIN {X 0,Y 543.664,Z 878.176,A -85,B 0,C 180,E1 22898.236,E2 22898.236} C_VEL
LIN {X 0,Y 546.649,Z 854.641,A -85,B 0,C 180,E1 22897.613,E2 22897.613} C_VEL
LIN {X 0,Y 549.424,Z 825.072,A -85,B 0,C 180,E1 22897.03,E2 22897.03} C_VEL
LIN {X 0,Y 552.677,Z 758.913,A -85,B 0,C 180,E1 22896.016,E2 22896.016} C_VEL
LIN {X 0,Y 563.246,Z 536.685,A -85,B 0,C 180,E1 22892.652,E2 22892.652} C_VEL
LIN {X 0,Y 566.776,Z 463.299,A -85,B 0,C 180,E1 22891.509,E2 22891.509} C_VEL
LIN {X 0,Y 555.027,Z 444.802,A -85,B 0,C 180,E1 22889.016,E2 22889.016} C_VEL
LIN {X 0,Y 545.084,Z 430.086,A -85,B 0,C 180,E1 22886.677,E2 22886.677} C_VEL
LIN {X 0,Y 535.272,Z 416.155,A -85,B 0,C 180,E1 22884.089,E2 22884.089} C_VEL
LIN {X 0,Y 527.733,Z 406.091,A -85,B 0,C 180,E1 22881.858,E2 22881.858} C_VEL
LIN {X 0,Y 523.292,Z 400.295,A -85,B 0,C 180,E1 22880.409,E2 22880.409} C_VEL
LIN {X 0,Y 518.293,Z 393.808,A -85,B 0,C 180,E1 22878.62,E2 22878.62} C_VEL
LIN {X 0,Y 515.938,Z 390.977,A -85,B 0,C 180,E1 22877.714,E2 22877.714} C_VEL
LIN {X 0,Y 512.668,Z 387.178,A -85,B 0,C 180,E1 22876.369,E2 22876.369} C_VEL
LIN {X 0,Y 511.598,Z 385.496,A -85,B 0,C 180,E1 22875.88,E2 22875.88} C_VEL
LIN {X 0,Y 508.022,Z 382.245,A -85,B 0,C 180,E1 22874.243,E2 22874.243} C_VEL
LIN {X 0,Y 506.212,Z 379.17,A -85,B 0,C 180,E1 22873.246,E2 22873.246} C_VEL
LIN {X 0,Y 502.897,Z 376.841,A -85,B 0,C 180,E1 22871.41,E2 22871.41} C_VEL
LIN {X 0,Y 500.718,Z 373.019,A -85,B 0,C 180,E1 22869.831,E2 22869.831} C_VEL
LIN {X 0,Y 500.019,Z 372.448,A -85,B 0,C 180,E1 22869.322,E2 22869.322} C_VEL
LIN {X 0,Y 496.246,Z 369.712,A -85,B 0,C 180,E1 22865.898,E2 22865.898} C_VEL
LIN {X 0,Y 494.793,Z 366.03,A -85,B 0,C 180,E1 22863.302,E2 22863.302} C_VEL
LIN {X 0,Y 494.778,Z 365.967,A -85,B 0,C 180,E1 22856.234,E2 22856.234} C_VEL
LIN {X 0,Y 496.039,Z 369.384,A -85,B 0,C 180,E1 22853.867,E2 22853.867} C_VEL
LIN {X 0,Y 499.645,Z 372.335,A -85,B 0,C 180,E1 22850.439,E2 22850.439} C_VEL
LIN {X 0,Y 500.665,Z 372.936,A -85,B 0,C 180,E1 22849.703,E2 22849.703} C_VEL
LIN {X 0,Y 502.481,Z 376.384,A -85,B 0,C 180,E1 22848.347,E2 22848.347} C_VEL
LIN {X 0,Y 506.13,Z 379.164,A -85,B 0,C 180,E1 22846.286,E2 22846.286} C_VEL
LIN {X 0,Y 509.051,Z 383.552,A -85,B 0,C 180,E1 22844.74,E2 22844.74} C_VEL
LIN {X 0,Y 511.931,Z 385.992,A -85,B 0,C 180,E1 22843.46,E2 22843.46} C_VEL
LIN {X 0,Y 515.016,Z 390.137,A -85,B 0,C 180,E1 22842.136,E2 22842.136} C_VEL
LIN {X 0,Y 517.323,Z 392.274,A -85,B 0,C 180,E1 22841.256,E2 22841.256} C_VEL
LIN {X 0,Y 520.979,Z 396.84,A -85,B 0,C 180,E1 22839.907,E2 22839.907} C_VEL
LIN {X 0,Y 522.728,Z 398.844,A -85,B 0,C 180,E1 22839.305,E2 22839.305} C_VEL
LIN {X 0,Y 527.745,Z 404.911,A -85,B 0,C 180,E1 22837.674,E2 22837.674} C_VEL
LIN {X 0,Y 532.329,Z 410.564,A -85,B 0,C 180,E1 22836.299,E2 22836.299} C_VEL
LIN {X 0,Y 537.251,Z 416.825,A -85,B 0,C 180,E1 22834.921,E2 22834.921} C_VEL
LIN {X 0,Y 544.307,Z 425.667,A -85,B 0,C 180,E1 22833.105,E2 22833.105} C_VEL
LIN {X 0,Y 555.343,Z 440.553,A -85,B 0,C 180,E1 22830.529,E2 22830.529} C_VEL
LIN {X 0,Y 566.784,Z 456.772,A -85,B 0,C 180,E1 22828.137,E2 22828.137} C_VEL
LIN {X 0,Y 556.463,Z 666.547,A -85,B 0,C 180,E1 22824.946,E2 22824.946} C_VEL
LIN {X 0,Y 549.982,Z 801.279,A -85,B 0,C 180,E1 22822.9,E2 22822.9} C_VEL
LIN {X 0,Y 547.822,Z 826.78,A -85,B 0,C 180,E1 22822.411,E2 22822.411} C_VEL
LIN {X 0,Y 544.537,Z 854.272,A -85,B 0,C 180,E1 22821.69,E2 22821.69} C_VEL
LIN {X 0,Y 541.413,Z 875.685,A -85,B 0,C 180,E1 22820.985,E2 22820.985} C_VEL
LIN {X 0,Y 538.084,Z 895.552,A -85,B 0,C 180,E1 22820.206,E2 22820.206} C_VEL
LIN {X 0,Y 534.266,Z 915.771,A -85,B 0,C 180,E1 22819.283,E2 22819.283} C_VEL
LIN {X 0,Y 529.729,Z 937.539,A -85,B 0,C 180,E1 22818.126,E2 22818.126} C_VEL
LIN {X 0,Y 523.726,Z 963.259,A -85,B 0,C 180,E1 22816.507,E2 22816.507} C_VEL
LIN {X 0,Y 518.836,Z 982.591,A -85,B 0,C 180,E1 22815.09,E2 22815.09} C_VEL
LIN {X 0,Y 514.04,Z 1000.61,A -85,B 0,C 180,E1 22813.593,E2 22813.593} C_VEL
LIN {X 0,Y 509.138,Z 1018.31,A -85,B 0,C 180,E1 22811.936,E2 22811.936} C_VEL
LIN {X 0,Y 503.229,Z 1038.953,A -85,B 0,C 180,E1 22809.74,E2 22809.74} C_VEL
LIN {X 0,Y 498.709,Z 1054.35,A -85,B 0,C 180,E1 22807.861,E2 22807.861} C_VEL
LIN {X 0,Y 496.315,Z 1059.589,A -85,B 0,C 180,E1 22807.249,E2 22807.249} C_VEL
LIN {X 0,Y 487.398,Z 1072.894,A -85,B 0,C 180,E1 22805.829,E2 22805.829} C_VEL
LIN {X 0,Y 485.154,Z 1077.719,A -85,B 0,C 180,E1 22805.175,E2 22805.175} C_VEL
LIN {X 0,Y 480.076,Z 1094.448,A -85,B 0,C 180,E1 22802.361,E2 22802.361} C_VEL
LIN {X 0,Y 476.454,Z 1106.98,A -85,B 0,C 180,E1 22799.964,E2 22799.964} C_VEL
LIN {X 0,Y 473.338,Z 1118.518,A -85,B 0,C 180,E1 22797.474,E2 22797.474} C_VEL
LIN {X 0,Y 470.215,Z 1131.182,A -85,B 0,C 180,E1 22794.363,E2 22794.363} C_VEL
LIN {X 0,Y 467.797,Z 1142.039,A -85,B 0,C 180,E1 22791.175,E2 22791.175} C_VEL
LIN {X 0,Y 466.318,Z 1149.877,A -85,B 0,C 180,E1 22788.502,E2 22788.502} C_VEL
LIN {X 0,Y 465.324,Z 1156.267,A -85,B 0,C 180,E1 22785.964,E2 22785.964} C_VEL
LIN {X 0,Y 464.634,Z 1161.899,A -85,B 0,C 180,E1 22783.312,E2 22783.312} C_VEL
LIN {X 0,Y 464.199,Z 1166.871,A -85,B 0,C 180,E1 22780.424,E2 22780.424} C_VEL
LIN {X 0,Y 463.978,Z 1171.231,A -85,B 0,C 180,E1 22777.056,E2 22777.056} C_VEL
LIN {X 0,Y 463.917,Z 1173.649,A -85,B 0,C 180,E1 22774.079,E2 22774.079} C_VEL
LIN {X 0,Y 463.908,Z 1174.726,A -85,B 0,C 180,E1 22771.482,E2 22771.482} C_VEL
LIN {X 0,Y 463.906,Z 1174.833,A -85,B 0,C 180,E1 22769.012,E2 22769.012} C_VEL
LIN {X 0,Y 463.914,Z 1173.972,A -85,B 0,C 180,E1 22766.417,E2 22766.417} C_VEL
LIN {X 0,Y 463.952,Z 1172.11,A -85,B 0,C 180,E1 22763.814,E2 22763.814} C_VEL
LIN {X 0,Y 464.051,Z 1169.398,A -85,B 0,C 180,E1 22761.325,E2 22761.325} C_VEL
LIN {X 0,Y 464.304,Z 1165.264,A -85,B 0,C 180,E1 22758.481,E2 22758.481} C_VEL
LIN {X 0,Y 464.897,Z 1159.603,A -85,B 0,C 180,E1 22755.426,E2 22755.426} C_VEL
LIN {X 0,Y 466.048,Z 1151.497,A -85,B 0,C 180,E1 22752.005,E2 22752.005} C_VEL
LIN {X 0,Y 467.497,Z 1143.497,A -85,B 0,C 180,E1 22749.205,E2 22749.205} C_VEL
LIN {X 0,Y 469.265,Z 1135.075,A -85,B 0,C 180,E1 22746.652,E2 22746.652} C_VEL
LIN {X 0,Y 471.678,Z 1124.971,A -85,B 0,C 180,E1 22743.973,E2 22743.973} C_VEL
LIN {X 0,Y 475.359,Z 1111.116,A -85,B 0,C 180,E1 22740.792,E2 22740.792} C_VEL
LIN {X 0,Y 479.134,Z 1097.639,A -85,B 0,C 180,E1 22738.132,E2 22738.132} C_VEL
LIN {X 0,Y 482.956,Z 1084.723,A -85,B 0,C 180,E1 22735.872,E2 22735.872} C_VEL
LIN {X 0,Y 487.069,Z 1071.194,A -85,B 0,C 180,E1 22733.757,E2 22733.757} C_VEL
LIN {X 0,Y 492.26,Z 1054.391,A -85,B 0,C 180,E1 22731.423,E2 22731.423} C_VEL
LIN {X 0,Y 498.508,Z 1033.814,A -85,B 0,C 180,E1 22728.953,E2 22728.953} C_VEL
LIN {X 0,Y 503.59,Z 1016.679,A -85,B 0,C 180,E1 22727.155,E2 22727.155} C_VEL
LIN {X 0,Y 508.281,Z 1000.359,A -85,B 0,C 180,E1 22725.628,E2 22725.628} C_VEL
LIN {X 0,Y 513.268,Z 982.279,A -85,B 0,C 180,E1 22724.123,E2 22724.123} C_VEL
LIN {X 0,Y 518.984,Z 960.457,A -85,B 0,C 180,E1 22722.531,E2 22722.531} C_VEL
LIN {X 0,Y 524.77,Z 935.966,A -85,B 0,C 180,E1 22721.018,E2 22721.018} C_VEL
LIN {X 0,Y 529.239,Z 915.081,A -85,B 0,C 180,E1 22719.912,E2 22719.912} C_VEL
LIN {X 0,Y 533.178,Z 894.724,A -85,B 0,C 180,E1 22718.986,E2 22718.986} C_VEL
LIN {X 0,Y 536.882,Z 873.142,A -85,B 0,C 180,E1 22718.152,E2 22718.152} C_VEL
LIN {X 0,Y 540.845,Z 845.635,A -85,B 0,C 180,E1 22717.291,E2 22717.291} C_VEL
LIN {X 0,Y 543.537,Z 821.343,A -85,B 0,C 180,E1 22716.706,E2 22716.706} C_VEL
LIN {X 0,Y 545.386,Z 799.192,A -85,B 0,C 180,E1 22716.297,E2 22716.297} C_VEL
LIN {X 0,Y 556.035,Z 585.224,A -85,B 0,C 180,E1 22713.04,E2 22713.04} C_VEL
LIN {X 0,Y 562.366,Z 461.219,A -85,B 0,C 180,E1 22711.128,E2 22711.128} C_VEL
LIN {X 0,Y 551.382,Z 445.573,A -85,B 0,C 180,E1 22708.752,E2 22708.752} C_VEL
LIN {X 0,Y 540.988,Z 431.54,A -85,B 0,C 180,E1 22706.244,E2 22706.244} C_VEL
LIN {X 0,Y 532.599,Z 420.815,A -85,B 0,C 180,E1 22703.982,E2 22703.982} C_VEL
LIN {X 0,Y 528.129,Z 415.196,A -85,B 0,C 180,E1 22702.661,E2 22702.661} C_VEL
LIN {X 0,Y 524.059,Z 410.16,A -85,B 0,C 180,E1 22701.372,E2 22701.372} C_VEL
LIN {X 0,Y 519.478,Z 404.566,A -85,B 0,C 180,E1 22699.802,E2 22699.802} C_VEL
LIN {X 0,Y 515.659,Z 399.842,A -85,B 0,C 180,E1 22698.367,E2 22698.367} C_VEL
LIN {X 0,Y 511.31,Z 395.15,A -85,B 0,C 180,E1 22696.589,E2 22696.589} C_VEL
LIN {X 0,Y 509.893,Z 393.095,A -85,B 0,C 180,E1 22695.935,E2 22695.935} C_VEL
LIN {X 0,Y 506.537,Z 389.888,A -85,B 0,C 180,E1 22694.344,E2 22694.344} C_VEL
LIN {X 0,Y 504.873,Z 387.006,A -85,B 0,C 180,E1 22693.398,E2 22693.398} C_VEL
LIN {X 0,Y 501.141,Z 384.037,A -85,B 0,C 180,E1 22691.218,E2 22691.218} C_VEL
LIN {X 0,Y 499.329,Z 380.532,A -85,B 0,C 180,E1 22689.8,E2 22689.8} C_VEL
LIN {X 0,Y 495.529,Z 377.952,A -85,B 0,C 180,E1 22686.372,E2 22686.372} C_VEL
LIN {X 0,Y 493.858,Z 374.343,A -85,B 0,C 180,E1 22683.366,E2 22683.366} C_VEL
LIN {X 0,Y 493.626,Z 373.836,A -85,B 0,C 180,E1 22682.67,E2 22682.67} C_VEL
LIN {X 0,Y 493.863,Z 374.121,A -85,B 0,C 180,E1 22677.099,E2 22677.099} C_VEL
LIN {X 0,Y 495.303,Z 377.728,A -85,B 0,C 180,E1 22674.323,E2 22674.323} C_VEL
LIN {X 0,Y 499.108,Z 380.421,A -85,B 0,C 180,E1 22670.777,E2 22670.777} C_VEL
LIN {X 0,Y 499.544,Z 380.956,A -85,B 0,C 180,E1 22670.437,E2 22670.437} C_VEL
LIN {X 0,Y 501.842,Z 384.819,A -85,B 0,C 180,E1 22668.74,E2 22668.74} C_VEL
LIN {X 0,Y 505.099,Z 387.38,A -85,B 0,C 180,E1 22666.887,E2 22666.887} C_VEL
LIN {X 0,Y 507.763,Z 391.271,A -85,B 0,C 180,E1 22665.459,E2 22665.459} C_VEL
LIN {X 0,Y 510.578,Z 393.832,A -85,B 0,C 180,E1 22664.175,E2 22664.175} C_VEL
LIN {X 0,Y 513.749,Z 398.061,A -85,B 0,C 180,E1 22662.792,E2 22662.792} C_VEL
LIN {X 0,Y 515.654,Z 400.058,A -85,B 0,C 180,E1 22662.042,E2 22662.042} C_VEL
LIN {X 0,Y 520.098,Z 405.953,A -85,B 0,C 180,E1 22660.369,E2 22660.369} C_VEL
LIN {X 0,Y 523.743,Z 410.739,A -85,B 0,C 180,E1 22659.113,E2 22659.113} C_VEL
LIN {X 0,Y 528.337,Z 416.914,A -85,B 0,C 180,E1 22657.642,E2 22657.642} C_VEL
LIN {X 0,Y 534.987,Z 426.135,A -85,B 0,C 180,E1 22655.692,E2 22655.692} C_VEL
LIN {X 0,Y 543.875,Z 438.841,A -85,B 0,C 180,E1 22653.347,E2 22653.347} C_VEL
LIN {X 0,Y 554.603,Z 455.14,A -85,B 0,C 180,E1 22650.811,E2 22650.811} C_VEL
LIN {X 0,Y 562.515,Z 468.107,A -85,B 0,C 180,E1 22649.096,E2 22649.096} C_VEL
LIN {X 0,Y 551.853,Z 678.975,A -85,B 0,C 180,E1 22645.876,E2 22645.876} C_VEL
LIN {X 0,Y 544.784,Z 822.718,A -85,B 0,C 180,E1 22643.684,E2 22643.684} C_VEL
LIN {X 0,Y 542.406,Z 849.408,A -85,B 0,C 180,E1 22643.181,E2 22643.181} C_VEL
LIN {X 0,Y 538.959,Z 876.301,A -85,B 0,C 180,E1 22642.491,E2 22642.491} C_VEL
LIN {X 0,Y 535.647,Z 897.835,A -85,B 0,C 180,E1 22641.799,E2 22641.799} C_VEL
LIN {X 0,Y 532.009,Z 918.624,A -85,B 0,C 180,E1 22640.998,E2 22640.998} C_VEL
LIN {X 0,Y 527.899,Z 939.566,A -85,B 0,C 180,E1 22640.051,E2 22640.051} C_VEL
LIN {X 0,Y 522.413,Z 964.979,A -85,B 0,C 180,E1 22638.695,E2 22638.695} C_VEL
LIN {X 0,Y 516.809,Z 988.051,A -85,B 0,C 180,E1 22637.227,E2 22637.227} C_VEL
LIN {X 0,Y 511.991,Z 1006.774,A -85,B 0,C 180,E1 22635.863,E2 22635.863} C_VEL
LIN {X 0,Y 507.212,Z 1024.47,A -85,B 0,C 180,E1 22634.411,E2 22634.411} C_VEL
LIN {X 0,Y 502.202,Z 1042.379,A -85,B 0,C 180,E1 22632.759,E2 22632.759} C_VEL
LIN {X 0,Y 496.242,Z 1063.305,A -85,B 0,C 180,E1 22630.568,E2 22630.568} C_VEL
LIN {X 0,Y 490.451,Z 1082.869,A -85,B 0,C 180,E1 22628.187,E2 22628.187} C_VEL
LIN {X 0,Y 486.176,Z 1097.559,A -85,B 0,C 180,E1 22626.174,E2 22626.174} C_VEL
LIN {X 0,Y 482.18,Z 1111.491,A -85,B 0,C 180,E1 22624.047,E2 22624.047} C_VEL
LIN {X 0,Y 478.294,Z 1125.541,A -85,B 0,C 180,E1 22621.648,E2 22621.648} C_VEL
LIN {X 0,Y 473.938,Z 1142.187,A -85,B 0,C 180,E1 22618.385,E2 22618.385} C_VEL
LIN {X 0,Y 471.19,Z 1153.671,A -85,B 0,C 180,E1 22615.786,E2 22615.786} C_VEL
LIN {X 0,Y 469.018,Z 1163.671,A -85,B 0,C 180,E1 22613.228,E2 22613.228} C_VEL
LIN {X 0,Y 467.32,Z 1172.463,A -85,B 0,C 180,E1 22610.673,E2 22610.673} C_VEL
LIN {X 0,Y 465.939,Z 1180.835,A -85,B 0,C 180,E1 22607.87,E2 22607.87} C_VEL
LIN {X 0,Y 464.832,Z 1189.576,A -85,B 0,C 180,E1 22604.322,E2 22604.322} C_VEL
LIN {X 0,Y 464.291,Z 1195.213,A -85,B 0,C 180,E1 22601.427,E2 22601.427} C_VEL
LIN {X 0,Y 464.067,Z 1199.021,A -85,B 0,C 180,E1 22598.924,E2 22598.924} C_VEL
LIN {X 0,Y 463.958,Z 1201.842,A -85,B 0,C 180,E1 22596.434,E2 22596.434} C_VEL
LIN {X 0,Y 463.915,Z 1203.743,A -85,B 0,C 180,E1 22593.955,E2 22593.955} C_VEL
LIN {X 0,Y 463.911,Z 1204.734,A -85,B 0,C 180,E1 22591.482,E2 22591.482} C_VEL
LIN {X 0,Y 463.908,Z 1204.825,A -85,B 0,C 180,E1 22589.012,E2 22589.012} C_VEL
LIN {X 0,Y 463.915,Z 1204.015,A -85,B 0,C 180,E1 22586.54,E2 22586.54} C_VEL
LIN {X 0,Y 463.947,Z 1202.181,A -85,B 0,C 180,E1 22583.938,E2 22583.938} C_VEL
LIN {X 0,Y 464.043,Z 1199.499,A -85,B 0,C 180,E1 22581.45,E2 22581.45} C_VEL
LIN {X 0,Y 464.236,Z 1196.063,A -85,B 0,C 180,E1 22579.075,E2 22579.075} C_VEL
LIN {X 0,Y 464.662,Z 1191.145,A -85,B 0,C 180,E1 22576.435,E2 22576.435} C_VEL
LIN {X 0,Y 465.317,Z 1185.285,A -85,B 0,C 180,E1 22573.85,E2 22573.85} C_VEL
LIN {X 0,Y 466.399,Z 1177.936,A -85,B 0,C 180,E1 22571.113,E2 22571.113} C_VEL
LIN {X 0,Y 468.282,Z 1167.427,A -85,B 0,C 180,E1 22567.795,E2 22567.795} C_VEL
LIN {X 0,Y 470.707,Z 1155.783,A -85,B 0,C 180,E1 22564.726,E2 22564.726} C_VEL
LIN {X 0,Y 473.171,Z 1145.321,A -85,B 0,C 180,E1 22562.297,E2 22562.297} C_VEL
LIN {X 0,Y 476.124,Z 1133.611,A -85,B 0,C 180,E1 22559.874,E2 22559.874} C_VEL
LIN {X 0,Y 479.671,Z 1120.549,A -85,B 0,C 180,E1 22557.467,E2 22557.467} C_VEL
LIN {X 0,Y 484.739,Z 1102.648,A -85,B 0,C 180,E1 22554.566,E2 22554.566} C_VEL
LIN {X 0,Y 489.553,Z 1085.923,A -85,B 0,C 180,E1 22552.214,E2 22552.214} C_VEL
LIN {X 0,Y 494.114,Z 1070.265,A -85,B 0,C 180,E1 22550.25,E2 22550.25} C_VEL
LIN {X 0,Y 498.996,Z 1053.454,A -85,B 0,C 180,E1 22548.368,E2 22548.368} C_VEL
LIN {X 0,Y 505.119,Z 1032.172,A -85,B 0,C 180,E1 22546.263,E2 22546.263} C_VEL
LIN {X 0,Y 510.999,Z 1010.44,A -85,B 0,C 180,E1 22544.424,E2 22544.424} C_VEL
LIN {X 0,Y 515.866,Z 991.63,A -85,B 0,C 180,E1 22543.022,E2 22543.022} C_VEL
LIN {X 0,Y 520.619,Z 972.187,A -85,B 0,C 180,E1 22541.745,E2 22541.745} C_VEL
LIN {X 0,Y 525.272,Z 951.861,A -85,B 0,C 180,E1 22540.58,E2 22540.58} C_VEL
LIN {X 0,Y 530.595,Z 926.281,A -85,B 0,C 180,E1 22539.326,E2 22539.326} C_VEL
LIN {X 0,Y 535.027,Z 901.448,A -85,B 0,C 180,E1 22538.333,E2 22538.333} C_VEL
LIN {X 0,Y 538.402,Z 879.861,A -85,B 0,C 180,E1 22537.618,E2 22537.618} C_VEL
LIN {X 0,Y 541.233,Z 858.59,A -85,B 0,C 180,E1 22537.04,E2 22537.04} C_VEL
LIN {X 0,Y 543.807,Z 834.811,A -85,B 0,C 180,E1 22536.531,E2 22536.531} C_VEL
LIN {X 0,Y 546.079,Z 798.767,A -85,B 0,C 180,E1 22535.94,E2 22535.94} C_VEL
LIN {X 0,Y 556.876,Z 576.887,A -85,B 0,C 180,E1 22532.574,E2 22532.574} C_VEL
LIN {X 0,Y 562.397,Z 467.742,A -85,B 0,C 180,E1 22530.889,E2 22530.889} C_VEL
LIN {X 0,Y 551.819,Z 450.925,A -85,B 0,C 180,E1 22528.579,E2 22528.579} C_VEL
LIN {X 0,Y 542.335,Z 436.684,A -85,B 0,C 180,E1 22526.292,E2 22526.292} C_VEL
LIN {X 0,Y 532.857,Z 423.079,A -85,B 0,C 180,E1 22523.735,E2 22523.735} C_VEL
LIN {X 0,Y 525.607,Z 413.257,A -85,B 0,C 180,E1 22521.54,E2 22521.54} C_VEL
LIN {X 0,Y 521.392,Z 407.66,A -85,B 0,C 180,E1 22520.135,E2 22520.135} C_VEL
LIN {X 0,Y 516.472,Z 401.179,A -85,B 0,C 180,E1 22518.337,E2 22518.337} C_VEL
LIN {X 0,Y 514.147,Z 398.432,A -85,B 0,C 180,E1 22517.427,E2 22517.427} C_VEL
LIN {X 0,Y 510.833,Z 394.342,A -85,B 0,C 180,E1 22516.021,E2 22516.021} C_VEL
LIN {X 0,Y 509.878,Z 393.059,A -85,B 0,C 180,E1 22515.585,E2 22515.585} C_VEL
LIN {X 0,Y 506.293,Z 389.497,A -85,B 0,C 180,E1 22513.884,E2 22513.884} C_VEL
LIN {X 0,Y 504.817,Z 386.959,A -85,B 0,C 180,E1 22513.05,E2 22513.05} C_VEL
LIN {X 0,Y 501.484,Z 384.429,A -85,B 0,C 180,E1 22511.152,E2 22511.152} C_VEL
LIN {X 0,Y 499.216,Z 380.458,A -85,B 0,C 180,E1 22509.453,E2 22509.453} C_VEL
LIN {X 0,Y 495.362,Z 377.839,A -85,B 0,C 180,E1 22506.025,E2 22506.025} C_VEL
LIN {X 0,Y 493.761,Z 373.951,A -85,B 0,C 180,E1 22503.192,E2 22503.192} C_VEL
LIN {X 0,Y 493.769,Z 373.96,A -85,B 0,C 180,E1 22496.285,E2 22496.285} C_VEL
LIN {X 0,Y 494.975,Z 377.263,A -85,B 0,C 180,E1 22493.97,E2 22493.97} C_VEL
LIN {X 0,Y 498.529,Z 380.227,A -85,B 0,C 180,E1 22490.534,E2 22490.534} C_VEL
LIN {X 0,Y 499.448,Z 380.855,A -85,B 0,C 180,E1 22489.853,E2 22489.853} C_VEL
LIN {X 0,Y 501.42,Z 384.389,A -85,B 0,C 180,E1 22488.381,E2 22488.381} C_VEL
LIN {X 0,Y 505.04,Z 387.333,A -85,B 0,C 180,E1 22486.315,E2 22486.315} C_VEL
LIN {X 0,Y 507.625,Z 391.243,A -85,B 0,C 180,E1 22484.929,E2 22484.929} C_VEL
LIN {X 0,Y 510.457,Z 393.778,A -85,B 0,C 180,E1 22483.645,E2 22483.645} C_VEL
LIN {X 0,Y 513.65,Z 397.955,A -85,B 0,C 180,E1 22482.263,E2 22482.263} C_VEL
LIN {X 0,Y 515.718,Z 399.968,A -85,B 0,C 180,E1 22481.46,E2 22481.46} C_VEL
LIN {X 0,Y 519.568,Z 404.672,A -85,B 0,C 180,E1 22480.026,E2 22480.026} C_VEL
LIN {X 0,Y 525.946,Z 412.511,A -85,B 0,C 180,E1 22477.888,E2 22477.888} C_VEL
LIN {X 0,Y 530.395,Z 418.066,A -85,B 0,C 180,E1 22476.531,E2 22476.531} C_VEL
LIN {X 0,Y 535.175,Z 424.211,A -85,B 0,C 180,E1 22475.171,E2 22475.171} C_VEL
LIN {X 0,Y 542.056,Z 432.969,A -85,B 0,C 180,E1 22473.369,E2 22473.369} C_VEL
LIN {X 0,Y 552.663,Z 447.441,A -85,B 0,C 180,E1 22470.848,E2 22470.848} C_VEL
LIN {X 0,Y 562.375,Z 461.456,A -85,B 0,C 180,E1 22468.76,E2 22468.76} C_VEL
LIN {X 0,Y 551.455,Z 675.969,A -85,B 0,C 180,E1 22465.488,E2 22465.488} C_VEL
LIN {X 0,Y 545.18,Z 801.738,A -85,B 0,C 180,E1 22463.568,E2 22463.568} C_VEL
LIN {X 0,Y 542.88,Z 828.069,A -85,B 0,C 180,E1 22463.06,E2 22463.06} C_VEL
LIN {X 0,Y 539.531,Z 854.98,A -85,B 0,C 180,E1 22462.346,E2 22462.346} C_VEL
LIN {X 0,Y 536.352,Z 876.13,A -85,B 0,C 180,E1 22461.647,E2 22461.647} C_VEL
LIN {X 0,Y 532.948,Z 895.827,A -85,B 0,C 180,E1 22460.874,E2 22460.874} C_VEL
LIN {X 0,Y 529.016,Z 916.045,A -85,B 0,C 180,E1 22459.948,E2 22459.948} C_VEL
LIN {X 0,Y 524.338,Z 937.813,A -85,B 0,C 180,E1 22458.787,E2 22458.787} C_VEL
LIN {X 0,Y 518.138,Z 963.533,A -85,B 0,C 180,E1 22457.163,E2 22457.163} C_VEL
LIN {X 0,Y 513.102,Z 982.793,A -85,B 0,C 180,E1 22455.744,E2 22455.744} C_VEL
LIN {X 0,Y 508.2,Z 1000.578,A -85,B 0,C 180,E1 22454.26,E2 22454.26} C_VEL
LIN {X 0,Y 503.265,Z 1017.755,A -85,B 0,C 180,E1 22452.647,E2 22452.647} C_VEL
LIN {X 0,Y 497.429,Z 1037.495,A -85,B 0,C 180,E1 22450.551,E2 22450.551} C_VEL
LIN {X 0,Y 491.551,Z 1056.566,A -85,B 0,C 180,E1 22448.196,E2 22448.196} C_VEL
LIN {X 0,Y 486.97,Z 1071.505,A -85,B 0,C 180,E1 22446.105,E2 22446.105} C_VEL
LIN {X 0,Y 485.154,Z 1077.719,A -85,B 0,C 180,E1 22445.175,E2 22445.175} C_VEL
LIN {X 0,Y 482.897,Z 1082.502,A -85,B 0,C 180,E1 22444.501,E2 22444.501} C_VEL
LIN {X 0,Y 473.573,Z 1095.098,A -85,B 0,C 180,E1 22442.779,E2 22442.779} C_VEL
LIN {X 0,Y 471.799,Z 1098.806,A -85,B 0,C 180,E1 22442.145,E2 22442.145} C_VEL
LIN {X 0,Y 467.169,Z 1114.531,A -85,B 0,C 180,E1 22438.927,E2 22438.927} C_VEL
LIN {X 0,Y 464.028,Z 1125.925,A -85,B 0,C 180,E1 22436.214,E2 22436.214} C_VEL
LIN {X 0,Y 461.61,Z 1135.526,A -85,B 0,C 180,E1 22433.614,E2 22433.614} C_VEL
LIN {X 0,Y 459.753,Z 1143.893,A -85,B 0,C 180,E1 22431.029,E2 22431.029} C_VEL
LIN {X 0,Y 458.207,Z 1151.871,A -85,B 0,C 180,E1 22428.182,E2 22428.182} C_VEL
LIN {X 0,Y 456.947,Z 1160.192,A -85,B 0,C 180,E1 22424.574,E2 22424.574} C_VEL
LIN {X 0,Y 456.351,Z 1165.534,A -85,B 0,C 180,E1 22421.629,E2 22421.629} C_VEL
LIN {X 0,Y 456.084,Z 1169.35,A -85,B 0,C 180,E1 22418.955,E2 22418.955} C_VEL
LIN {X 0,Y 455.962,Z 1172.165,A -85,B 0,C 180,E1 22416.295,E2 22416.295} C_VEL
LIN {X 0,Y 455.916,Z 1173.959,A -85,B 0,C 180,E1 22413.725,E2 22413.725} C_VEL
LIN {X 0,Y 455.909,Z 1174.846,A -85,B 0,C 180,E1 22411.131,E2 22411.131} C_VEL
LIN {X 0,Y 455.908,Z 1174.819,A -85,B 0,C 180,E1 22408.618,E2 22408.618} C_VEL
LIN {X 0,Y 455.919,Z 1173.85,A -85,B 0,C 180,E1 22405.976,E2 22405.976} C_VEL
LIN {X 0,Y 455.966,Z 1171.914,A -85,B 0,C 180,E1 22403.326,E2 22403.326} C_VEL
LIN {X 0,Y 456.124,Z 1168.687,A -85,B 0,C 180,E1 22400.41,E2 22400.41} C_VEL
LIN {X 0,Y 456.61,Z 1163.083,A -85,B 0,C 180,E1 22396.836,E2 22396.836} C_VEL
LIN {X 0,Y 457.373,Z 1157.038,A -85,B 0,C 180,E1 22393.881,E2 22393.881} C_VEL
LIN {X 0,Y 458.479,Z 1150.387,A -85,B 0,C 180,E1 22391.17,E2 22391.17} C_VEL
LIN {X 0,Y 460.034,Z 1142.579,A -85,B 0,C 180,E1 22388.45,E2 22388.45} C_VEL
LIN {X 0,Y 462.575,Z 1131.758,A -85,B 0,C 180,E1 22385.208,E2 22385.208} C_VEL
LIN {X 0,Y 465.799,Z 1119.379,A -85,B 0,C 180,E1 22382.099,E2 22382.099} C_VEL
LIN {X 0,Y 469.124,Z 1107.651,A -85,B 0,C 180,E1 22379.519,E2 22379.519} C_VEL
LIN {X 0,Y 472.698,Z 1095.846,A -85,B 0,C 180,E1 22377.215,E2 22377.215} C_VEL
LIN {X 0,Y 477.32,Z 1081.205,A -85,B 0,C 180,E1 22374.68,E2 22374.68} C_VEL
LIN {X 0,Y 483.378,Z 1062.095,A -85,B 0,C 180,E1 22371.818,E2 22371.818} C_VEL
LIN {X 0,Y 488.277,Z 1046.679,A -85,B 0,C 180,E1 22369.803,E2 22369.803} C_VEL
LIN {X 0,Y 493.304,Z 1030.694,A -85,B 0,C 180,E1 22367.943,E2 22367.943} C_VEL
LIN {X 0,Y 498.644,Z 1013.341,A -85,B 0,C 180,E1 22366.15,E2 22366.15} C_VEL
LIN {X 0,Y 505.113,Z 991.484,A -85,B 0,C 180,E1 22364.171,E2 22364.171} C_VEL
LIN {X 0,Y 511.106,Z 969.564,A -85,B 0,C 180,E1 22362.48,E2 22362.48} C_VEL
LIN {X 0,Y 516.088,Z 950.188,A -85,B 0,C 180,E1 22361.178,E2 22361.178} C_VEL
LIN {X 0,Y 520.735,Z 930.721,A -85,B 0,C 180,E1 22360.035,E2 22360.035} C_VEL
LIN {X 0,Y 525.576,Z 908.273,A -85,B 0,C 180,E1 22358.889,E2 22358.889} C_VEL
LIN {X 0,Y 530.552,Z 881.655,A -85,B 0,C 180,E1 22357.771,E2 22357.771} C_VEL
LIN {X 0,Y 534.03,Z 859.866,A -85,B 0,C 180,E1 22357.021,E2 22357.021} C_VEL
LIN {X 0,Y 536.894,Z 838.485,A -85,B 0,C 180,E1 22356.414,E2 22356.414} C_VEL
LIN {X 0,Y 539.279,Z 816.633,A -85,B 0,C 180,E1 22355.922,E2 22355.922} C_VEL
LIN {X 0,Y 541.401,Z 788.427,A -85,B 0,C 180,E1 22355.433,E2 22355.433} C_VEL
LIN {X 0,Y 552.775,Z 565.155,A -85,B 0,C 180,E1 22352.031,E2 22352.031} C_VEL
LIN {X 0,Y 558.048,Z 465.961,A -85,B 0,C 180,E1 22350.499,E2 22350.499} C_VEL
LIN {X 0,Y 548.636,Z 452.314,A -85,B 0,C 180,E1 22348.403,E2 22348.403} C_VEL
LIN {X 0,Y 538.481,Z 438.451,A -85,B 0,C 180,E1 22345.902,E2 22345.902} C_VEL
LIN {X 0,Y 530.217,Z 427.768,A -85,B 0,C 180,E1 22343.624,E2 22343.624} C_VEL
LIN {X 0,Y 525.987,Z 422.373,A -85,B 0,C 180,E1 22342.346,E2 22342.346} C_VEL
LIN {X 0,Y 521.979,Z 417.373,A -85,B 0,C 180,E1 22341.049,E2 22341.049} C_VEL
LIN {X 0,Y 517.623,Z 411.973,A -85,B 0,C 180,E1 22339.523,E2 22339.523} C_VEL
LIN {X 0,Y 513.188,Z 406.542,A -85,B 0,C 180,E1 22337.812,E2 22337.812} C_VEL
LIN {X 0,Y 509.603,Z 402.517,A -85,B 0,C 180,E1 22336.295,E2 22336.295} C_VEL
LIN {X 0,Y 508.442,Z 400.817,A -85,B 0,C 180,E1 22335.747,E2 22335.747} C_VEL
LIN {X 0,Y 505.033,Z 397.434,A -85,B 0,C 180,E1 22334.095,E2 22334.095} C_VEL
LIN {X 0,Y 503.49,Z 394.785,A -85,B 0,C 180,E1 22333.202,E2 22333.202} C_VEL
LIN {X 0,Y 499.836,Z 391.731,A -85,B 0,C 180,E1 22331.014,E2 22331.014} C_VEL
LIN {X 0,Y 498.05,Z 388.375,A -85,B 0,C 180,E1 22329.592,E2 22329.592} C_VEL
LIN {X 0,Y 494.191,Z 385.527,A -85,B 0,C 180,E1 22325.923,E2 22325.923} C_VEL
LIN {X 0,Y 492.695,Z 381.785,A -85,B 0,C 180,E1 22322.792,E2 22322.792} C_VEL
LIN {X 0,Y 492.84,Z 382.024,A -85,B 0,C 180,E1 22317.209,E2 22317.209} C_VEL
LIN {X 0,Y 494.414,Z 385.853,A -85,B 0,C 180,E1 22314.196,E2 22314.196} C_VEL
LIN {X 0,Y 498.274,Z 388.666,A -85,B 0,C 180,E1 22310.645,E2 22310.645} C_VEL
LIN {X 0,Y 500.693,Z 392.715,A -85,B 0,C 180,E1 22308.831,E2 22308.831} C_VEL
LIN {X 0,Y 503.696,Z 395.081,A -85,B 0,C 180,E1 22307.096,E2 22307.096} C_VEL
LIN {X 0,Y 506.454,Z 399.077,A -85,B 0,C 180,E1 22305.596,E2 22305.596} C_VEL
LIN {X 0,Y 509.054,Z 401.5,A -85,B 0,C 180,E1 22304.389,E2 22304.389} C_VEL
LIN {X 0,Y 512.385,Z 405.874,A -85,B 0,C 180,E1 22302.921,E2 22302.921} C_VEL
LIN {X 0,Y 514.533,Z 408.326,A -85,B 0,C 180,E1 22302.06,E2 22302.06} C_VEL
LIN {X 0,Y 521.072,Z 416.959,A -85,B 0,C 180,E1 22299.647,E2 22299.647} C_VEL
LIN {X 0,Y 528.441,Z 427.083,A -85,B 0,C 180,E1 22297.265,E2 22297.265} C_VEL
LIN {X 0,Y 535.975,Z 437.961,A -85,B 0,C 180,E1 22295.093,E2 22295.093} C_VEL
LIN {X 0,Y 543.84,Z 449.526,A -85,B 0,C 180,E1 22293.05,E2 22293.05} C_VEL
LIN {X 0,Y 553.153,Z 464.089,A -85,B 0,C 180,E1 22290.846,E2 22290.846} C_VEL
LIN {X 0,Y 558.162,Z 472.54,A -85,B 0,C 180,E1 22289.734,E2 22289.734} C_VEL
LIN {X 0,Y 547.136,Z 683.475,A -85,B 0,C 180,E1 22286.502,E2 22286.502} C_VEL
LIN {X 0,Y 540.056,Z 822.473,A -85,B 0,C 180,E1 22284.372,E2 22284.372} C_VEL
LIN {X 0,Y 537.602,Z 849.291,A -85,B 0,C 180,E1 22283.865,E2 22283.865} C_VEL
LIN {X 0,Y 534.064,Z 876.075,A -85,B 0,C 180,E1 22283.179,E2 22283.179} C_VEL
LIN {X 0,Y 530.66,Z 897.576,A -85,B 0,C 180,E1 22282.489,E2 22282.489} C_VEL
LIN {X 0,Y 526.916,Z 918.362,A -85,B 0,C 180,E1 22281.687,E2 22281.687} C_VEL
LIN {X 0,Y 522.789,Z 938.749,A -85,B 0,C 180,E1 22280.767,E2 22280.767} C_VEL
LIN {X 0,Y 517.498,Z 962.694,A -85,B 0,C 180,E1 22279.497,E2 22279.497} C_VEL
LIN {X 0,Y 511.479,Z 986.831,A -85,B 0,C 180,E1 22277.974,E2 22277.974} C_VEL
LIN {X 0,Y 506.438,Z 1005.762,A -85,B 0,C 180,E1 22276.597,E2 22276.597} C_VEL
LIN {X 0,Y 501.481,Z 1023.463,A -85,B 0,C 180,E1 22275.144,E2 22275.144} C_VEL
LIN {X 0,Y 496.355,Z 1041.118,A -85,B 0,C 180,E1 22273.514,E2 22273.514} C_VEL
LIN {X 0,Y 490.587,Z 1060.568,A -85,B 0,C 180,E1 22271.481,E2 22271.481} C_VEL
LIN {X 0,Y 484.248,Z 1081.34,A -85,B 0,C 180,E1 22268.969,E2 22268.969} C_VEL
LIN {X 0,Y 479.428,Z 1097.163,A -85,B 0,C 180,E1 22266.787,E2 22266.787} C_VEL
LIN {X 0,Y 475.206,Z 1111.216,A -85,B 0,C 180,E1 22264.617,E2 22264.617} C_VEL
LIN {X 0,Y 470.985,Z 1125.724,A -85,B 0,C 180,E1 22262.105,E2 22262.105} C_VEL
LIN {X 0,Y 466.487,Z 1142.11,A -85,B 0,C 180,E1 22258.833,E2 22258.833} C_VEL
LIN {X 0,Y 463.504,Z 1153.921,A -85,B 0,C 180,E1 22256.108,E2 22256.108} C_VEL
LIN {X 0,Y 461.234,Z 1163.867,A -85,B 0,C 180,E1 22253.507,E2 22253.507} C_VEL
LIN {X 0,Y 459.386,Z 1173.019,A -85,B 0,C 180,E1 22250.779,E2 22250.779} C_VEL
LIN {X 0,Y 457.743,Z 1182.853,A -85,B 0,C 180,E1 22247.334,E2 22247.334} C_VEL
LIN {X 0,Y 456.801,Z 1190.092,A -85,B 0,C 180,E1 22244.191,E2 22244.191} C_VEL
LIN {X 0,Y 456.3,Z 1195.158,A -85,B 0,C 180,E1 22241.502,E2 22241.502} C_VEL
LIN {X 0,Y 456.068,Z 1198.98,A -85,B 0,C 180,E1 22238.955,E2 22238.955} C_VEL
LIN {X 0,Y 455.958,Z 1201.839,A -85,B 0,C 180,E1 22236.421,E2 22236.421} C_VEL
LIN {X 0,Y 455.914,Z 1203.752,A -85,B 0,C 180,E1 22233.898,E2 22233.898} C_VEL
LIN {X 0,Y 455.912,Z 1204.73,A -85,B 0,C 180,E1 22231.382,E2 22231.382} C_VEL
LIN {X 0,Y 455.911,Z 1204.777,A -85,B 0,C 180,E1 22228.869,E2 22228.869} C_VEL
LIN {X 0,Y 455.914,Z 1203.892,A -85,B 0,C 180,E1 22226.354,E2 22226.354} C_VEL
LIN {X 0,Y 455.949,Z 1202.072,A -85,B 0,C 180,E1 22223.832,E2 22223.832} C_VEL
LIN {X 0,Y 456.053,Z 1199.308,A -85,B 0,C 180,E1 22221.299,E2 22221.299} C_VEL
LIN {X 0,Y 456.268,Z 1195.583,A -85,B 0,C 180,E1 22218.753,E2 22218.753} C_VEL
LIN {X 0,Y 456.743,Z 1190.615,A -85,B 0,C 180,E1 22216.066,E2 22216.066} C_VEL
LIN {X 0,Y 457.43,Z 1184.844,A -85,B 0,C 180,E1 22213.492,E2 22213.492} C_VEL
LIN {X 0,Y 458.625,Z 1177.301,A -85,B 0,C 180,E1 22210.648,E2 22210.648} C_VEL
LIN {X 0,Y 460.757,Z 1166.216,A -85,B 0,C 180,E1 22207.143,E2 22207.143} C_VEL
LIN {X 0,Y 463.132,Z 1155.507,A -85,B 0,C 180,E1 22204.282,E2 22204.282} C_VEL
LIN {X 0,Y 465.71,Z 1145.044,A -85,B 0,C 180,E1 22201.814,E2 22201.814} C_VEL
LIN {X 0,Y 468.844,Z 1133.334,A -85,B 0,C 180,E1 22199.357,E2 22199.357} C_VEL
LIN {X 0,Y 472.794,Z 1119.558,A -85,B 0,C 180,E1 22196.789,E2 22196.789} C_VEL
LIN {X 0,Y 478.343,Z 1100.713,A -85,B 0,C 180,E1 22193.734,E2 22193.734} C_VEL
LIN {X 0,Y 483.193,Z 1084.704,A -85,B 0,C 180,E1 22191.475,E2 22191.475} C_VEL
LIN {X 0,Y 488.045,Z 1068.77,A -85,B 0,C 180,E1 22189.473,E2 22189.473} C_VEL
LIN {X 0,Y 493.792,Z 1049.865,A -85,B 0,C 180,E1 22187.366,E2 22187.366} C_VEL
LIN {X 0,Y 500.446,Z 1027.098,A -85,B 0,C 180,E1 22185.177,E2 22185.177} C_VEL
LIN {X 0,Y 505.763,Z 1008.142,A -85,B 0,C 180,E1 22183.592,E2 22183.592} C_VEL
LIN {X 0,Y 510.599,Z 990.047,A -85,B 0,C 180,E1 22182.252,E2 22182.252} C_VEL
LIN {X 0,Y 515.573,Z 970.261,A -85,B 0,C 180,E1 22180.959,E2 22180.959} C_VEL
LIN {X 0,Y 521.387,Z 945.486,A -85,B 0,C 180,E1 22179.564,E2 22179.564} C_VEL
LIN {X 0,Y 526.437,Z 920.706,A -85,B 0,C 180,E1 22178.413,E2 22178.413} C_VEL
LIN {X 0,Y 530.271,Z 899.673,A -85,B 0,C 180,E1 22177.589,E2 22177.589} C_VEL
LIN {X 0,Y 533.663,Z 878.497,A -85,B 0,C 180,E1 22176.897,E2 22176.897} C_VEL
LIN {X 0,Y 536.62,Z 856.64,A -85,B 0,C 180,E1 22176.31,E2 22176.31} C_VEL
LIN {X 0,Y 539.602,Z 828.625,A -85,B 0,C 180,E1 22175.733,E2 22175.733} C_VEL
LIN {X 0,Y 542.171,Z 782.402,A -85,B 0,C 180,E1 22175.005,E2 22175.005} C_VEL
LIN {X 0,Y 553.438,Z 560.079,A -85,B 0,C 180,E1 22171.616,E2 22171.616} C_VEL
LIN {X 0,Y 558.093,Z 472.214,A -85,B 0,C 180,E1 22170.261,E2 22170.261} C_VEL
LIN {X 0,Y 548.228,Z 456.399,A -85,B 0,C 180,E1 22168.038,E2 22168.038} C_VEL
LIN {X 0,Y 539.234,Z 442.706,A -85,B 0,C 180,E1 22165.804,E2 22165.804} C_VEL
LIN {X 0,Y 530.202,Z 429.656,A -85,B 0,C 180,E1 22163.301,E2 22163.301} C_VEL
LIN {X 0,Y 523.498,Z 420.421,A -85,B 0,C 180,E1 22161.22,E2 22161.22} C_VEL
LIN {X 0,Y 519.204,Z 414.653,A -85,B 0,C 180,E1 22159.754,E2 22159.754} C_VEL
LIN {X 0,Y 514.527,Z 408.373,A -85,B 0,C 180,E1 22157.998,E2 22157.998} C_VEL
LIN {X 0,Y 512.506,Z 405.999,A -85,B 0,C 180,E1 22157.192,E2 22157.192} C_VEL
LIN {X 0,Y 509.13,Z 401.701,A -85,B 0,C 180,E1 22155.725,E2 22155.725} C_VEL
LIN {X 0,Y 508.174,Z 400.599,A -85,B 0,C 180,E1 22155.287,E2 22155.287} C_VEL
LIN {X 0,Y 504.686,Z 396.888,A -85,B 0,C 180,E1 22153.578,E2 22153.578} C_VEL
LIN {X 0,Y 503.429,Z 394.74,A -85,B 0,C 180,E1 22152.853,E2 22152.853} C_VEL
LIN {X 0,Y 500.165,Z 392.122,A -85,B 0,C 180,E1 22150.948,E2 22150.948} C_VEL
LIN {X 0,Y 497.932,Z 388.297,A -85,B 0,C 180,E1 22149.244,E2 22149.244} C_VEL
LIN {X 0,Y 494.111,Z 385.467,A -85,B 0,C 180,E1 22145.691,E2 22145.691} C_VEL
LIN {X 0,Y 492.656,Z 381.786,A -85,B 0,C 180,E1 22142.908,E2 22142.908} C_VEL
LIN {X 0,Y 492.742,Z 381.854,A -85,B 0,C 180,E1 22136.393,E2 22136.393} C_VEL
LIN {X 0,Y 493.999,Z 385.256,A -85,B 0,C 180,E1 22133.958,E2 22133.958} C_VEL
LIN {X 0,Y 497.565,Z 388.185,A -85,B 0,C 180,E1 22130.515,E2 22130.515} C_VEL
LIN {X 0,Y 498.238,Z 388.751,A -85,B 0,C 180,E1 22130.003,E2 22130.003} C_VEL
LIN {X 0,Y 500.274,Z 392.287,A -85,B 0,C 180,E1 22128.471,E2 22128.471} C_VEL
LIN {X 0,Y 503.653,Z 395.085,A -85,B 0,C 180,E1 22126.51,E2 22126.51} C_VEL
LIN {X 0,Y 506.43,Z 399.168,A -85,B 0,C 180,E1 22125.01,E2 22125.01} C_VEL
LIN {X 0,Y 508.933,Z 401.446,A -85,B 0,C 180,E1 22123.859,E2 22123.859} C_VEL
LIN {X 0,Y 512.287,Z 405.769,A -85,B 0,C 180,E1 22122.39,E2 22122.39} C_VEL
LIN {X 0,Y 514.121,Z 407.65,A -85,B 0,C 180,E1 22121.664,E2 22121.664} C_VEL
LIN {X 0,Y 518.16,Z 412.499,A -85,B 0,C 180,E1 22120.146,E2 22120.146} C_VEL
LIN {X 0,Y 524.235,Z 420.214,A -85,B 0,C 180,E1 22118.077,E2 22118.077} C_VEL
LIN {X 0,Y 528.472,Z 425.562,A -85,B 0,C 180,E1 22116.766,E2 22116.766} C_VEL
LIN {X 0,Y 536.14,Z 435.382,A -85,B 0,C 180,E1 22114.599,E2 22114.599} C_VEL
LIN {X 0,Y 544.797,Z 447.17,A -85,B 0,C 180,E1 22112.392,E2 22112.392} C_VEL
LIN {X 0,Y 553.788,Z 459.699,A -85,B 0,C 180,E1 22110.319,E2 22110.319} C_VEL
LIN {X 0,Y 558.014,Z 466.316,A -85,B 0,C 180,E1 22109.393,E2 22109.393} C_VEL
LIN {X 0,Y 546.737,Z 680.563,A -85,B 0,C 180,E1 22106.114,E2 22106.114} C_VEL
LIN {X 0,Y 540.461,Z 802.057,A -85,B 0,C 180,E1 22104.251,E2 22104.251} C_VEL
LIN {X 0,Y 538.072,Z 828.674,A -85,B 0,C 180,E1 22103.735,E2 22103.735} C_VEL
LIN {X 0,Y 534.627,Z 855.472,A -85,B 0,C 180,E1 22103.022,E2 22103.022} C_VEL
LIN {X 0,Y 531.432,Z 876.172,A -85,B 0,C 180,E1 22102.337,E2 22102.337} C_VEL
LIN {X 0,Y 527.888,Z 896.101,A -85,B 0,C 180,E1 22101.554,E2 22101.554} C_VEL
LIN {X 0,Y 523.841,Z 916.319,A -85,B 0,C 180,E1 22100.626,E2 22100.626} C_VEL
LIN {X 0,Y 519.021,Z 938.087,A -85,B 0,C 180,E1 22099.462,E2 22099.462} C_VEL
LIN {X 0,Y 512.62,Z 963.807,A -85,B 0,C 180,E1 22097.832,E2 22097.832} C_VEL
LIN {X 0,Y 507.343,Z 983.327,A -85,B 0,C 180,E1 22096.386,E2 22096.386} C_VEL
LIN {X 0,Y 502.443,Z 1000.5,A -85,B 0,C 180,E1 22094.946,E2 22094.946} C_VEL
LIN {X 0,Y 497.576,Z 1016.83,A -85,B 0,C 180,E1 22093.411,E2 22093.411} C_VEL
LIN {X 0,Y 492.332,Z 1033.87,A -85,B 0,C 180,E1 22091.612,E2 22091.612} C_VEL
LIN {X 0,Y 485.97,Z 1054.106,A -85,B 0,C 180,E1 22089.171,E2 22089.171} C_VEL
LIN {X 0,Y 480.537,Z 1070.951,A -85,B 0,C 180,E1 22086.816,E2 22086.816} C_VEL
LIN {X 0,Y 475.98,Z 1085.277,A -85,B 0,C 180,E1 22084.553,E2 22084.553} C_VEL
LIN {X 0,Y 471.799,Z 1098.806,A -85,B 0,C 180,E1 22082.145,E2 22082.145} C_VEL
LIN {X 0,Y 469.664,Z 1103.101,A -85,B 0,C 180,E1 22081.399,E2 22081.399} C_VEL
LIN {X 0,Y 460.69,Z 1114.411,A -85,B 0,C 180,E1 22079.474,E2 22079.474} C_VEL
LIN {X 0,Y 459.025,Z 1117.597,A -85,B 0,C 180,E1 22078.78,E2 22078.78} C_VEL
LIN {X 0,Y 456.025,Z 1128.214,A -85,B 0,C 180,E1 22076.149,E2 22076.149} C_VEL
LIN {X 0,Y 453.184,Z 1139.357,A -85,B 0,C 180,E1 22072.986,E2 22072.986} C_VEL
LIN {X 0,Y 450.916,Z 1149.455,A -85,B 0,C 180,E1 22069.537,E2 22069.537} C_VEL
LIN {X 0,Y 449.671,Z 1156.22,A -85,B 0,C 180,E1 22066.802,E2 22066.802} C_VEL
LIN {X 0,Y 448.873,Z 1161.696,A -85,B 0,C 180,E1 22064.183,E2 22064.183} C_VEL
LIN {X 0,Y 448.341,Z 1166.403,A -85,B 0,C 180,E1 22061.448,E2 22061.448} C_VEL
LIN {X 0,Y 448.083,Z 1170.08,A -85,B 0,C 180,E1 22058.728,E2 22058.728} C_VEL
LIN {X 0,Y 447.957,Z 1172.87,A -85,B 0,C 180,E1 22055.893,E2 22055.893} C_VEL
LIN {X 0,Y 447.913,Z 1174.858,A -85,B 0,C 180,E1 22052.559,E2 22052.559} C_VEL
LIN {X 0,Y 447.904,Z 1175.192,A -85,B 0,C 180,E1 22049.233,E2 22049.233} C_VEL
LIN {X 0,Y 447.92,Z 1174.377,A -85,B 0,C 180,E1 22046.417,E2 22046.417} C_VEL
LIN {X 0,Y 447.967,Z 1172.618,A -85,B 0,C 180,E1 22043.721,E2 22043.721} C_VEL
LIN {X 0,Y 448.092,Z 1169.88,A -85,B 0,C 180,E1 22041.014,E2 22041.014} C_VEL
LIN {X 0,Y 448.347,Z 1166.341,A -85,B 0,C 180,E1 22038.422,E2 22038.422} C_VEL
LIN {X 0,Y 448.854,Z 1161.865,A -85,B 0,C 180,E1 22035.816,E2 22035.816} C_VEL
LIN {X 0,Y 449.687,Z 1156.126,A -85,B 0,C 180,E1 22033.066,E2 22033.066} C_VEL
LIN {X 0,Y 451.122,Z 1148.52,A -85,B 0,C 180,E1 22030.015,E2 22030.015} C_VEL
LIN {X 0,Y 453.523,Z 1137.856,A -85,B 0,C 180,E1 22026.482,E2 22026.482} C_VEL
LIN {X 0,Y 456.07,Z 1128.029,A -85,B 0,C 180,E1 22023.714,E2 22023.714} C_VEL
LIN {X 0,Y 459.077,Z 1117.404,A -85,B 0,C 180,E1 22021.085,E2 22021.085} C_VEL
LIN {X 0,Y 462.763,Z 1105.431,A -85,B 0,C 180,E1 22018.475,E2 22018.475} C_VEL
LIN {X 0,Y 468.255,Z 1088.293,A -85,B 0,C 180,E1 22015.242,E2 22015.242} C_VEL
LIN {X 0,Y 473.175,Z 1073.397,A -85,B 0,C 180,E1 22012.819,E2 22012.819} C_VEL
LIN {X 0,Y 478.113,Z 1058.579,A -85,B 0,C 180,E1 22010.68,E2 22010.68} C_VEL
LIN {X 0,Y 484.092,Z 1040.644,A -85,B 0,C 180,E1 22008.393,E2 22008.393} C_VEL
LIN {X 0,Y 490.858,Z 1019.616,A -85,B 0,C 180,E1 22006.086,E2 22006.086} C_VEL
LIN {X 0,Y 496.244,Z 1002.21,A -85,B 0,C 180,E1 22004.417,E2 22004.417} C_VEL
LIN {X 0,Y 501.349,Z 984.989,A -85,B 0,C 180,E1 22002.952,E2 22002.952} C_VEL
LIN {X 0,Y 506.498,Z 966.61,A -85,B 0,C 180,E1 22001.568,E2 22001.568} C_VEL
LIN {X 0,Y 511.899,Z 945.984,A -85,B 0,C 180,E1 22000.208,E2 22000.208} C_VEL
LIN {X 0,Y 518.029,Z 920.086,A -85,B 0,C 180,E1 21998.761,E2 21998.761} C_VEL
LIN {X 0,Y 522.665,Z 897.791,A -85,B 0,C 180,E1 21997.719,E2 21997.719} C_VEL
LIN {X 0,Y 526.439,Z 877.329,A -85,B 0,C 180,E1 21996.908,E2 21996.908} C_VEL
LIN {X 0,Y 529.813,Z 856.164,A -85,B 0,C 180,E1 21996.203,E2 21996.203} C_VEL
LIN {X 0,Y 533.33,Z 829.763,A -85,B 0,C 180,E1 21995.495,E2 21995.495} C_VEL
LIN {X 0,Y 535.851,Z 802.652,A -85,B 0,C 180,E1 21994.966,E2 21994.966} C_VEL
LIN {X 0,Y 541.347,Z 700.284,A -85,B 0,C 180,E1 21993.387,E2 21993.387} C_VEL
LIN {X 0,Y 552.987,Z 485.506,A -85,B 0,C 180,E1 21990.092,E2 21990.092} C_VEL
LIN {X 0,Y 553.808,Z 470.609,A -85,B 0,C 180,E1 21989.859,E2 21989.859} C_VEL
LIN {X 0,Y 544.005,Z 456.332,A -85,B 0,C 180,E1 21987.593,E2 21987.593} C_VEL
LIN {X 0,Y 533.337,Z 441.713,A -85,B 0,C 180,E1 21984.832,E2 21984.832} C_VEL
LIN {X 0,Y 524.357,Z 430.111,A -85,B 0,C 180,E1 21982.183,E2 21982.183} C_VEL
LIN {X 0,Y 519.916,Z 424.578,A -85,B 0,C 180,E1 21980.724,E2 21980.724} C_VEL
LIN {X 0,Y 515.926,Z 419.522,A -85,B 0,C 180,E1 21979.295,E2 21979.295} C_VEL
LIN {X 0,Y 511.55,Z 414.122,A -85,B 0,C 180,E1 21977.577,E2 21977.577} C_VEL
LIN {X 0,Y 507.911,Z 409.882,A -85,B 0,C 180,E1 21975.998,E2 21975.998} C_VEL
LIN {X 0,Y 506.753,Z 408.363,A -85,B 0,C 180,E1 21975.449,E2 21975.449} C_VEL
LIN {X 0,Y 503.44,Z 404.829,A -85,B 0,C 180,E1 21973.788,E2 21973.788} C_VEL
LIN {X 0,Y 502.114,Z 402.557,A -85,B 0,C 180,E1 21973.004,E2 21973.004} C_VEL
LIN {X 0,Y 498.537,Z 399.424,A -85,B 0,C 180,E1 21970.809,E2 21970.809} C_VEL
LIN {X 0,Y 496.779,Z 396.211,A -85,B 0,C 180,E1 21969.383,E2 21969.383} C_VEL
LIN {X 0,Y 492.965,Z 393.186,A -85,B 0,C 180,E1 21965.587,E2 21965.587} C_VEL
LIN {X 0,Y 491.678,Z 389.717,A -85,B 0,C 180,E1 21962.681,E2 21962.681} C_VEL
LIN {X 0,Y 491.82,Z 389.923,A -85,B 0,C 180,E1 21957.32,E2 21957.32} C_VEL
LIN {X 0,Y 493.438,Z 393.847,A -85,B 0,C 180,E1 21954.185,E2 21954.185} C_VEL
LIN {X 0,Y 497.074,Z 396.53,A -85,B 0,C 180,E1 21950.798,E2 21950.798} C_VEL
LIN {X 0,Y 499.545,Z 400.608,A -85,B 0,C 180,E1 21948.921,E2 21948.921} C_VEL
LIN {X 0,Y 502.411,Z 402.995,A -85,B 0,C 180,E1 21947.237,E2 21947.237} C_VEL
LIN {X 0,Y 505.373,Z 407.108,A -85,B 0,C 180,E1 21945.623,E2 21945.623} C_VEL
LIN {X 0,Y 507.594,Z 409.256,A -85,B 0,C 180,E1 21944.578,E2 21944.578} C_VEL
LIN {X 0,Y 511.024,Z 413.686,A -85,B 0,C 180,E1 21943.05,E2 21943.05} C_VEL
LIN {X 0,Y 513.546,Z 416.775,A -85,B 0,C 180,E1 21942.025,E2 21942.025} C_VEL
LIN {X 0,Y 519.841,Z 425.361,A -85,B 0,C 180,E1 21939.685,E2 21939.685} C_VEL
LIN {X 0,Y 526.194,Z 434.097,A -85,B 0,C 180,E1 21937.604,E2 21937.604} C_VEL
LIN {X 0,Y 534.061,Z 445.652,A -85,B 0,C 180,E1 21935.293,E2 21935.293} C_VEL
LIN {X 0,Y 541.844,Z 457.36,A -85,B 0,C 180,E1 21933.239,E2 21933.239} C_VEL
LIN {X 0,Y 550.358,Z 470.818,A -85,B 0,C 180,E1 21931.19,E2 21931.19} C_VEL
LIN {X 0,Y 553.884,Z 476.873,A -85,B 0,C 180,E1 21930.384,E2 21930.384} C_VEL
LIN {X 0,Y 542.552,Z 686.658,A -85,B 0,C 180,E1 21927.159,E2 21927.159} C_VEL
LIN {X 0,Y 535.398,Z 822.335,A -85,B 0,C 180,E1 21925.071,E2 21925.071} C_VEL
LIN {X 0,Y 532.833,Z 849.599,A -85,B 0,C 180,E1 21924.554,E2 21924.554} C_VEL
LIN {X 0,Y 529.209,Z 876.114,A -85,B 0,C 180,E1 21923.871,E2 21923.871} C_VEL
LIN {X 0,Y 525.624,Z 898.061,A -85,B 0,C 180,E1 21923.165,E2 21923.165} C_VEL
LIN {X 0,Y 521.899,Z 918.101,A -85,B 0,C 180,E1 21922.39,E2 21922.39} C_VEL
LIN {X 0,Y 517.648,Z 938.487,A -85,B 0,C 180,E1 21921.469,E2 21921.469} C_VEL
LIN {X 0,Y 512.105,Z 962.805,A -85,B 0,C 180,E1 21920.176,E2 21920.176} C_VEL
LIN {X 0,Y 505.975,Z 986.563,A -85,B 0,C 180,E1 21918.67,E2 21918.67} C_VEL
LIN {X 0,Y 500.756,Z 1005.493,A -85,B 0,C 180,E1 21917.289,E2 21917.289} C_VEL
LIN {X 0,Y 495.6,Z 1023.252,A -85,B 0,C 180,E1 21915.824,E2 21915.824} C_VEL
LIN {X 0,Y 490.24,Z 1041.058,A -85,B 0,C 180,E1 21914.168,E2 21914.168} C_VEL
LIN {X 0,Y 483.978,Z 1061.419,A -85,B 0,C 180,E1 21912.017,E2 21912.017} C_VEL
LIN {X 0,Y 477.54,Z 1081.619,A -85,B 0,C 180,E1 21909.532,E2 21909.532} C_VEL
LIN {X 0,Y 472.654,Z 1097.008,A -85,B 0,C 180,E1 21907.382,E2 21907.382} C_VEL
LIN {X 0,Y 468.283,Z 1110.94,A -85,B 0,C 180,E1 21905.204,E2 21905.204} C_VEL
LIN {X 0,Y 463.978,Z 1124.987,A -85,B 0,C 180,E1 21902.745,E2 21902.745} C_VEL
LIN {X 0,Y 459.125,Z 1141.834,A -85,B 0,C 180,E1 21899.34,E2 21899.34} C_VEL
LIN {X 0,Y 456.097,Z 1153.119,A -85,B 0,C 180,E1 21896.705,E2 21896.705} C_VEL
LIN {X 0,Y 453.673,Z 1163.12,A -85,B 0,C 180,E1 21894.062,E2 21894.062} C_VEL
LIN {X 0,Y 451.778,Z 1171.916,A -85,B 0,C 180,E1 21891.418,E2 21891.418} C_VEL
LIN {X 0,Y 450.212,Z 1180.346,A -85,B 0,C 180,E1 21888.496,E2 21888.496} C_VEL
LIN {X 0,Y 448.954,Z 1189.037,A -85,B 0,C 180,E1 21884.84,E2 21884.84} C_VEL
LIN {X 0,Y 448.352,Z 1194.679,A -85,B 0,C 180,E1 21881.839,E2 21881.839} C_VEL
LIN {X 0,Y 448.087,Z 1198.55,A -85,B 0,C 180,E1 21879.245,E2 21879.245} C_VEL
LIN {X 0,Y 447.963,Z 1201.475,A -85,B 0,C 180,E1 21876.645,E2 21876.645} C_VEL
LIN {X 0,Y 447.919,Z 1203.419,A -85,B 0,C 180,E1 21874.096,E2 21874.096} C_VEL
LIN {X 0,Y 447.915,Z 1204.444,A -85,B 0,C 180,E1 21871.535,E2 21871.535} C_VEL
LIN {X 0,Y 447.914,Z 1204.538,A -85,B 0,C 180,E1 21868.977,E2 21868.977} C_VEL
LIN {X 0,Y 447.918,Z 1203.699,A -85,B 0,C 180,E1 21866.417,E2 21866.417} C_VEL
LIN {X 0,Y 447.951,Z 1201.925,A -85,B 0,C 180,E1 21863.85,E2 21863.85} C_VEL
LIN {X 0,Y 448.054,Z 1199.207,A -85,B 0,C 180,E1 21861.272,E2 21861.272} C_VEL
LIN {X 0,Y 448.275,Z 1195.529,A -85,B 0,C 180,E1 21858.681,E2 21858.681} C_VEL
LIN {X 0,Y 448.769,Z 1190.608,A -85,B 0,C 180,E1 21855.945,E2 21855.945} C_VEL
LIN {X 0,Y 449.487,Z 1184.885,A -85,B 0,C 180,E1 21853.324,E2 21853.324} C_VEL
LIN {X 0,Y 450.673,Z 1177.724,A -85,B 0,C 180,E1 21850.551,E2 21850.551} C_VEL
LIN {X 0,Y 452.669,Z 1167.766,A -85,B 0,C 180,E1 21847.261,E2 21847.261} C_VEL
LIN {X 0,Y 455.449,Z 1155.758,A -85,B 0,C 180,E1 21843.956,E2 21843.956} C_VEL
LIN {X 0,Y 458.333,Z 1144.616,A -85,B 0,C 180,E1 21841.282,E2 21841.282} C_VEL
LIN {X 0,Y 461.804,Z 1132.409,A -85,B 0,C 180,E1 21838.693,E2 21838.693} C_VEL
LIN {X 0,Y 466.631,Z 1116.414,A -85,B 0,C 180,E1 21835.7,E2 21835.7} C_VEL
LIN {X 0,Y 471.832,Z 1099.575,A -85,B 0,C 180,E1 21833,E2 21833} C_VEL
LIN {X 0,Y 476.624,Z 1084.425,A -85,B 0,C 180,E1 21830.844,E2 21830.844} C_VEL
LIN {X 0,Y 481.621,Z 1068.68,A -85,B 0,C 180,E1 21828.845,E2 21828.845} C_VEL
LIN {X 0,Y 487.289,Z 1050.711,A -85,B 0,C 180,E1 21826.819,E2 21826.819} C_VEL
LIN {X 0,Y 494.408,Z 1027.324,A -85,B 0,C 180,E1 21824.539,E2 21824.539} C_VEL
